REGION Network 24: Inicjacja parametrów nastwa zbirników z Modbus TCP
   RUNG wire#powerrail
      Move(in := "dbtags_Sterowanie"."Paramaetry _Zbiorniki".set_poziom_napełniania, out1 => "dbHold_RRG".set_poziom_napełniania)
      Move(in := "dbtags_Sterowanie"."Paramaetry _Zbiorniki".set_poziom_opróżniania, out1 => "dbHold_RRG".set_poziom_opróżniania)
      Move(in := "dbtags_Sterowanie"."Paramaetry _Zbiorniki".set_bity_sterowania_napęami_1, out1 => "dbHold_RRG".set_res_bity_sterowania_napęami_1)
      Move(in := "dbtags_Sterowanie"."Paramaetry _Zbiorniki".set_bity_sterowania_napęami_2, out1 => "dbHold_RRG".set_res_bity_sterowania_napęami_2)
      Move(in := "dbtags_Sterowanie"."Paramaetry _Zbiorniki".set_bity_tryb_napędów_1, out1 => "dbHold_RRG".set_res_bity_tryb_napędów_1)
      Move(in := "dbtags_Sterowanie"."Paramaetry _Zbiorniki".set_bity_tryb_napędów_2, out1 => "dbHold_RRG".set_res_bity_tryb_napędów_2)
   END_RUNG
   // the same network as SCL:
   "dbHold_RRG".set_poziom_napełniania := "dbtags_Sterowanie"."Paramaetry _Zbiorniki".set_poziom_napełniania;
   "dbHold_RRG".set_poziom_opróżniania := "dbtags_Sterowanie"."Paramaetry _Zbiorniki".set_poziom_opróżniania;
   "dbHold_RRG".set_res_bity_sterowania_napęami_1 := "dbtags_Sterowanie"."Paramaetry _Zbiorniki".set_bity_sterowania_napęami_1;
   "dbHold_RRG".set_res_bity_sterowania_napęami_2 := "dbtags_Sterowanie"."Paramaetry _Zbiorniki".set_bity_sterowania_napęami_2;
   "dbHold_RRG".set_res_bity_tryb_napędów_1 := "dbtags_Sterowanie"."Paramaetry _Zbiorniki".set_bity_tryb_napędów_1;
   "dbHold_RRG".set_res_bity_tryb_napędów_2 := "dbtags_Sterowanie"."Paramaetry _Zbiorniki".set_bity_tryb_napędów_2;
END_REGION

REGION Network 25
   RUNG wire#powerrail
      Move(in := "dbtags_Sterowanie"."Paramaetry _Zbiorniki".set_strategia_sterowania, out1 => "dbHold_RRG".set_strategia_sterowania)
      Move(in := "dbtags_Sterowanie"."Paramaetry _Zbiorniki".set_sterowanie_cyklem, out1 => "dbHold_RRG".set_sterowanie_cyklem)
      Move(in := "dbtags_Sterowanie"."Paramaetry _Zbiorniki".set_położenie_Z10, out1 => "dbHold_RRG".set_położenie_Z10)
   END_RUNG
   // the same network as SCL:
   "dbHold_RRG".set_strategia_sterowania := "dbtags_Sterowanie"."Paramaetry _Zbiorniki".set_strategia_sterowania;
   "dbHold_RRG".set_sterowanie_cyklem := "dbtags_Sterowanie"."Paramaetry _Zbiorniki".set_sterowanie_cyklem;
   "dbHold_RRG".set_położenie_Z10 := "dbtags_Sterowanie"."Paramaetry _Zbiorniki".set_położenie_Z10;
END_REGION

REGION Network 26: Napełnianie
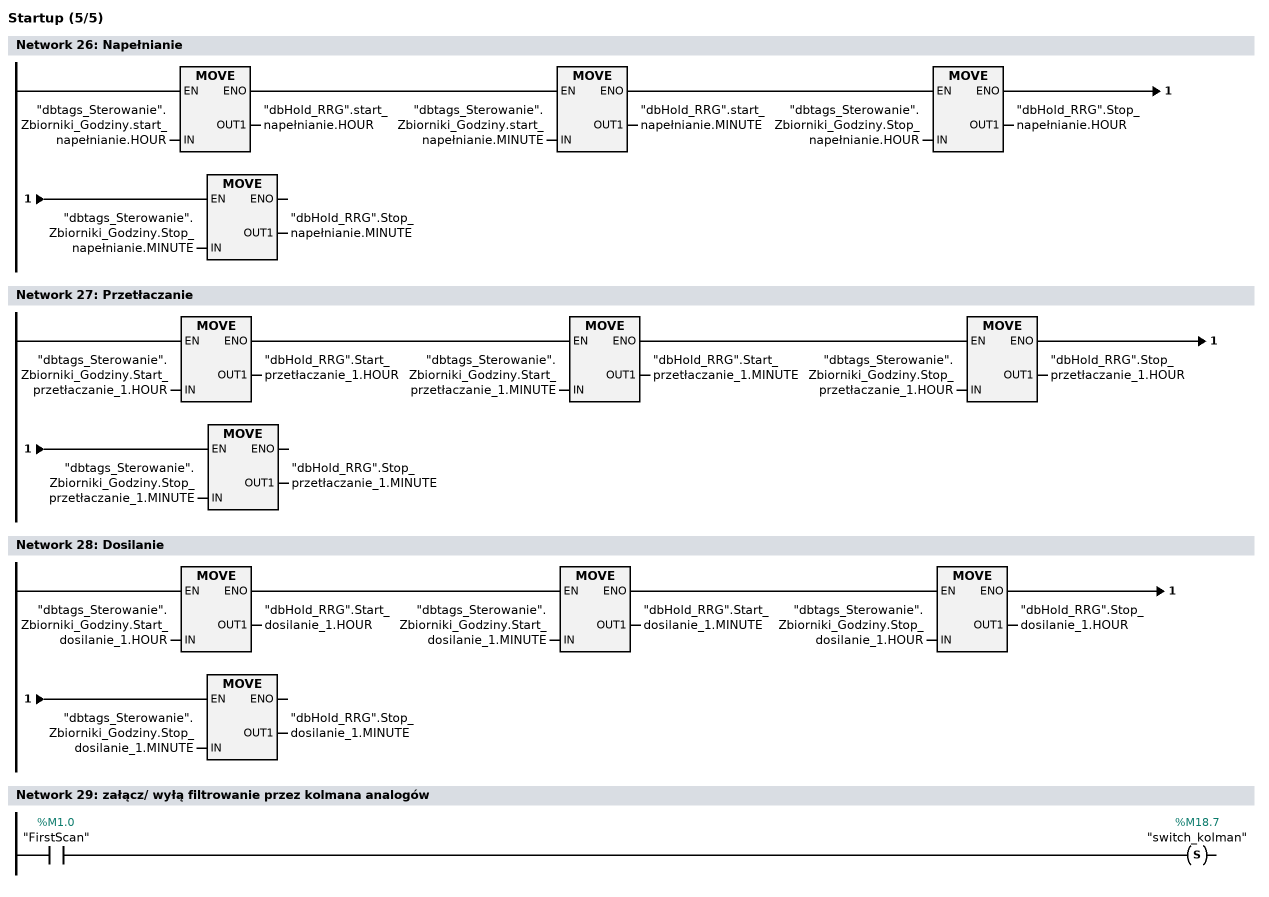
   RUNG wire#powerrail
      Move(in := "dbtags_Sterowanie".Zbiorniki_Godziny.start_napełnianie.HOUR, out1 => "dbHold_RRG".start_napełnianie.HOUR)
      Move(in := "dbtags_Sterowanie".Zbiorniki_Godziny.start_napełnianie.MINUTE, out1 => "dbHold_RRG".start_napełnianie.MINUTE)
      Move(in := "dbtags_Sterowanie".Zbiorniki_Godziny.Stop_napełnianie.HOUR, out1 => "dbHold_RRG".Stop_napełnianie.HOUR)
      Move(in := "dbtags_Sterowanie".Zbiorniki_Godziny.Stop_napełnianie.MINUTE, out1 => "dbHold_RRG".Stop_napełnianie.MINUTE)
   END_RUNG
   // the same network as SCL:
   "dbHold_RRG".start_napełnianie.HOUR := "dbtags_Sterowanie".Zbiorniki_Godziny.start_napełnianie.HOUR;
   "dbHold_RRG".start_napełnianie.MINUTE := "dbtags_Sterowanie".Zbiorniki_Godziny.start_napełnianie.MINUTE;
   "dbHold_RRG".Stop_napełnianie.HOUR := "dbtags_Sterowanie".Zbiorniki_Godziny.Stop_napełnianie.HOUR;
   "dbHold_RRG".Stop_napełnianie.MINUTE := "dbtags_Sterowanie".Zbiorniki_Godziny.Stop_napełnianie.MINUTE;
END_REGION

REGION Network 27: Przetłaczanie
   RUNG wire#powerrail
      Move(in := "dbtags_Sterowanie".Zbiorniki_Godziny.Start_przetłaczanie_1.HOUR, out1 => "dbHold_RRG".Start_przetłaczanie_1.HOUR)
      Move(in := "dbtags_Sterowanie".Zbiorniki_Godziny.Start_przetłaczanie_1.MINUTE, out1 => "dbHold_RRG".Start_przetłaczanie_1.MINUTE)
      Move(in := "dbtags_Sterowanie".Zbiorniki_Godziny.Stop_przetłaczanie_1.HOUR, out1 => "dbHold_RRG".Stop_przetłaczanie_1.HOUR)
      Move(in := "dbtags_Sterowanie".Zbiorniki_Godziny.Stop_przetłaczanie_1.MINUTE, out1 => "dbHold_RRG".Stop_przetłaczanie_1.MINUTE)
   END_RUNG
   // the same network as SCL:
   "dbHold_RRG".Start_przetłaczanie_1.HOUR := "dbtags_Sterowanie".Zbiorniki_Godziny.Start_przetłaczanie_1.HOUR;
   "dbHold_RRG".Start_przetłaczanie_1.MINUTE := "dbtags_Sterowanie".Zbiorniki_Godziny.Start_przetłaczanie_1.MINUTE;
   "dbHold_RRG".Stop_przetłaczanie_1.HOUR := "dbtags_Sterowanie".Zbiorniki_Godziny.Stop_przetłaczanie_1.HOUR;
   "dbHold_RRG".Stop_przetłaczanie_1.MINUTE := "dbtags_Sterowanie".Zbiorniki_Godziny.Stop_przetłaczanie_1.MINUTE;
END_REGION

REGION Network 28: Dosilanie
   RUNG wire#powerrail
      Move(in := "dbtags_Sterowanie".Zbiorniki_Godziny.Start_dosilanie_1.HOUR, out1 => "dbHold_RRG".Start_dosilanie_1.HOUR)
      Move(in := "dbtags_Sterowanie".Zbiorniki_Godziny.Start_dosilanie_1.MINUTE, out1 => "dbHold_RRG".Start_dosilanie_1.MINUTE)
      Move(in := "dbtags_Sterowanie".Zbiorniki_Godziny.Stop_dosilanie_1.HOUR, out1 => "dbHold_RRG".Stop_dosilanie_1.HOUR)
      Move(in := "dbtags_Sterowanie".Zbiorniki_Godziny.Stop_dosilanie_1.MINUTE, out1 => "dbHold_RRG".Stop_dosilanie_1.MINUTE)
   END_RUNG
   // the same network as SCL:
   "dbHold_RRG".Start_dosilanie_1.HOUR := "dbtags_Sterowanie".Zbiorniki_Godziny.Start_dosilanie_1.HOUR;
   "dbHold_RRG".Start_dosilanie_1.MINUTE := "dbtags_Sterowanie".Zbiorniki_Godziny.Start_dosilanie_1.MINUTE;
   "dbHold_RRG".Stop_dosilanie_1.HOUR := "dbtags_Sterowanie".Zbiorniki_Godziny.Stop_dosilanie_1.HOUR;
   "dbHold_RRG".Stop_dosilanie_1.MINUTE := "dbtags_Sterowanie".Zbiorniki_Godziny.Stop_dosilanie_1.MINUTE;
END_REGION

REGION Network 29: załącz/ wyłą filtrowanie przez kolmana analogów
   RUNG wire#powerrail
      Contact( "FirstScan" )
      S_Coil( "switch_kolman" )
   END_RUNG
   // the same network as SCL:
   IF "FirstScan" THEN "switch_kolman" := TRUE; END_IF;
END_REGION
END_ORGANIZATION_BLOCK

FUNCTION_BLOCK "Temp"   // FB22, LAD
{ S7_Optimized_Access := 'TRUE' }
VERSION : 0.1
// stored: AutoNumber true, IsIECCheckEnabled false, IsRetainMemResEnabled false, MemoryReserve 100, SetENOAutomatically false, UDAEnableTagReadback false
   VAR_INPUT
      Sub_PV_K1 : Real;   // Wspólczynnik pomniejszenia wyliczanego ciśnienia napotrzeby wyłączenia dodatowej pompy / Wspólczynnik pomniejszenia wyliczanego tlenu napotrzeby wyłączenia dodatowej dmuchawy
      InputWarning_H_PID { ExternalAccessible := 'False'; ExternalVisible := 'False'; ExternalWritable := 'False'} : Bool;   // Oszczerzenie górny limit
      InputWarning_L_PID { ExternalAccessible := 'False'; ExternalVisible := 'False'; ExternalWritable := 'False'} : Bool;   // Oczszczerzenie dolny limit
   END_VAR
   VAR_IN_OUT
      Set_K1 { ExternalWritable := 'False'} : Bool;   // Dostaw 1 dodatkową / Dostaw 1 dmuchawę dodatkową
   END_VAR
   VAR_TEMP
      Temp_SV_Int : Int;
   END_VAR
   VAR_TEMP   // added for the SCL form of the ladder/FBD networks
      _w1 : Bool;
      _w2 : Bool;
   END_VAR
BEGIN

REGION Network 1
   // OB 30 Network 14
END_REGION

REGION Network 2: Przekazanie wartości na wyjście analogowe "Out_Hz" -
   // Jeśli znacznik TmP_Set_SV (tymczasowe ustawienie Hz) wyłączony to na wyjście QW90 przekazywana jest wartość wyliczona z PID
   // Jeśli znacznik Tmp_Set_SV jest True to na wyjście przekazywana jest wartość tymczasowa 30Hz
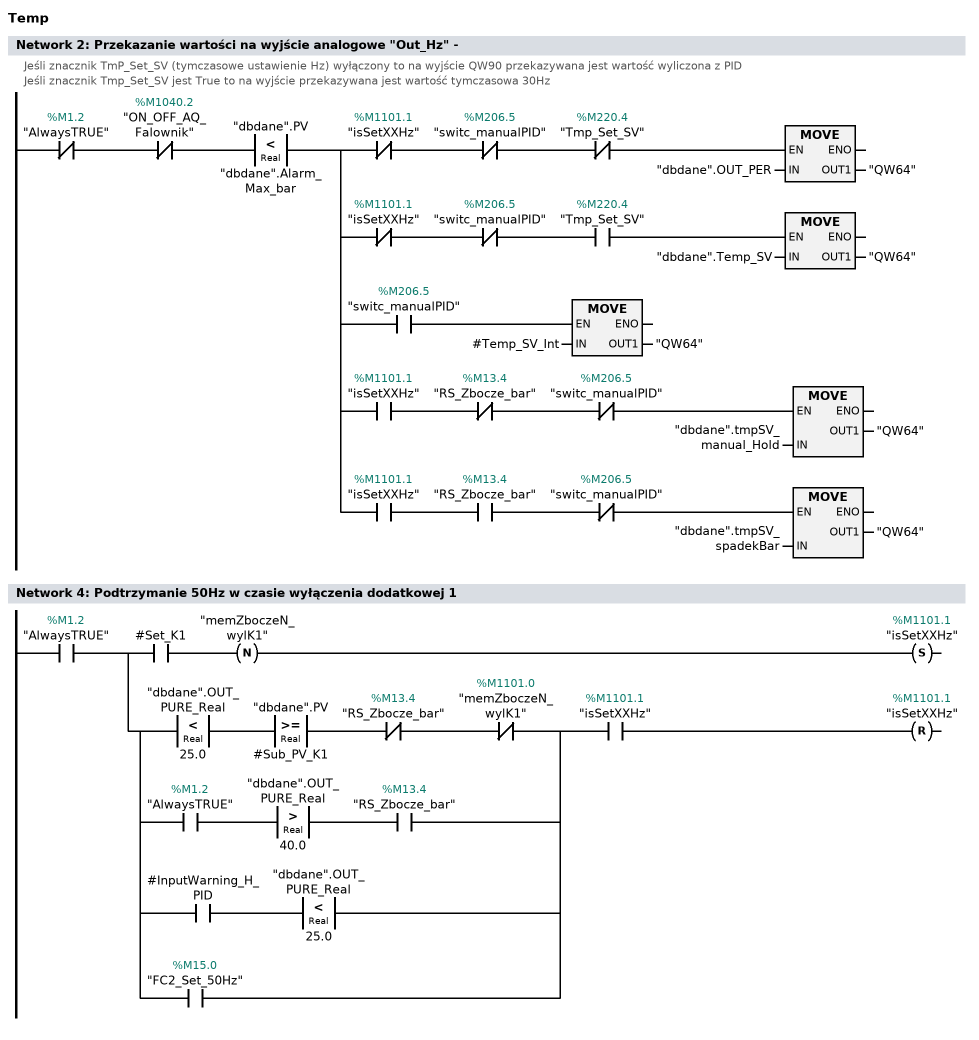
   RUNG wire#powerrail
      I_Contact( "AlwaysTRUE" )
      I_Contact( "ON_OFF_AQ_Falownik" )
      { S7_Templates := "SrcType := Real" } LT_Contact(in1 := "dbdane".PV, in2 := "dbdane".Alarm_Max_bar)
      wire#w1
      I_Contact( "isSetXXHz" )
      I_Contact( "switc_manualPID" )
      I_Contact( "Tmp_Set_SV" )
      { S7_GenerateENO := "TRUE" } Move(in := "dbdane".OUT_PER, out1 => "QW64")
   END_RUNG
   RUNG wire#w1
      I_Contact( "isSetXXHz" )
      I_Contact( "switc_manualPID" )
      Contact( "Tmp_Set_SV" )
      { S7_GenerateENO := "TRUE" } Move(in := "dbdane".Temp_SV, out1 => "QW64")
   END_RUNG
   RUNG wire#w1
      Contact( "switc_manualPID" )
      { S7_GenerateENO := "TRUE" } Move(in := #Temp_SV_Int, out1 => "QW64")
   END_RUNG
   RUNG wire#w1
      Contact( "isSetXXHz" )
      I_Contact( "RS_Zbocze_bar" )
      I_Contact( "switc_manualPID" )
      { S7_GenerateENO := "TRUE" } Move(in := "dbdane".tmpSV_manual_Hold, out1 => "QW64")
   END_RUNG
   RUNG wire#w1
      Contact( "isSetXXHz" )
      Contact( "RS_Zbocze_bar" )
      I_Contact( "switc_manualPID" )
      { S7_GenerateENO := "TRUE" } Move(in := "dbdane".tmpSV_spadekBar, out1 => "QW64")
   END_RUNG
   // the same network as SCL:
   #_w1 := NOT "AlwaysTRUE" AND NOT "ON_OFF_AQ_Falownik" AND ("dbdane".PV < "dbdane".Alarm_Max_bar);
   IF #_w1 AND NOT "isSetXXHz" AND NOT "switc_manualPID" AND NOT "Tmp_Set_SV" THEN
       "QW64" := "dbdane".OUT_PER;
   END_IF;
   IF #_w1 AND NOT "isSetXXHz" AND NOT "switc_manualPID" AND "Tmp_Set_SV" THEN
       "QW64" := "dbdane".Temp_SV;
   END_IF;
   IF #_w1 AND "switc_manualPID" THEN "QW64" := #Temp_SV_Int; END_IF;
   IF #_w1 AND "isSetXXHz" AND NOT "RS_Zbocze_bar" AND NOT "switc_manualPID" THEN
       "QW64" := "dbdane".tmpSV_manual_Hold;
   END_IF;
   IF #_w1 AND "isSetXXHz" AND "RS_Zbocze_bar" AND NOT "switc_manualPID" THEN
       "QW64" := "dbdane".tmpSV_spadekBar;
   END_IF;
END_REGION

REGION Network 3: FB1 Network 22
END_REGION

REGION Network 4: Podtrzymanie 50Hz w czasie wyłączenia dodatkowej 1
   RUNG wire#powerrail
      Contact( "AlwaysTRUE" )
      wire#w1
      Contact( #Set_K1 )
      N_Trig( "memZboczeN_wylK1" )
      S_Coil( "isSetXXHz" )
   END_RUNG
   RUNG wire#w1
      { S7_Templates := "SrcType := Real" } LT_Contact(in1 := "dbdane".OUT_PURE_Real, in2 := 25.0)
      { S7_Templates := "SrcType := Real" } GE_Contact(in1 := "dbdane".PV, in2 := #Sub_PV_K1)
      I_Contact( "RS_Zbocze_bar" )
      I_Contact( "memZboczeN_wylK1" )
      wire#w2
      Contact( "isSetXXHz" )
      R_Coil( "isSetXXHz" )
   END_RUNG
   RUNG wire#w1
      Contact( "AlwaysTRUE" )
      { S7_Templates := "SrcType := Real" } GT_Contact(in1 := "dbdane".OUT_PURE_Real, in2 := 40.0)
      Contact( "RS_Zbocze_bar" )
   END_RUNG wire#w2
   RUNG wire#w1
      Contact( #InputWarning_H_PID )
      { S7_Templates := "SrcType := Real" } LT_Contact(in1 := "dbdane".OUT_PURE_Real, in2 := 25.0)
   END_RUNG wire#w2
   RUNG wire#w1
      Contact( "FC2_Set_50Hz" )
   END_RUNG wire#w2
   // the same network as SCL:
   #_w1 := "AlwaysTRUE" AND #Set_K1;
   #_w2 := NOT #_w1 AND "memZboczeN_wylK1";   // falling edge
   "memZboczeN_wylK1" := #_w1;
   IF #_w2 THEN "isSetXXHz" := TRUE; END_IF;
   IF "AlwaysTRUE" AND ((("dbdane".OUT_PURE_Real < 25.0) AND ("dbdane".PV >= #Sub_PV_K1) AND NOT "RS_Zbocze_bar" AND NOT "memZboczeN_wylK1") OR ("AlwaysTRUE" AND ("dbdane".OUT_PURE_Real > 40.0) AND "RS_Zbocze_bar") OR (#InputWarning_H_PID AND ("dbdane".OUT_PURE_Real < 25.0)) OR "FC2_Set_50Hz") AND "isSetXXHz" THEN
       "isSetXXHz" := FALSE;
   END_IF;
END_REGION
END_FUNCTION_BLOCK

FUNCTION_BLOCK "WatchDog PLC - WinCC"   // FB13, LAD
TITLE = WatchDog PLC - WinCC
{ S7_Optimized_Access := 'TRUE' }
AUTHOR : rtecmer
VERSION : 0.1
// Kontrola komunikacji PLC z WinCC SCADA . Zerwanie komunikacji przekazywane do WinCC SCADA i PLC Master S7-300 (RS3)
// stored: AutoNumber true, IsIECCheckEnabled false, IsRetainMemResEnabled false, MemoryReserve 500, SetENOAutomatically false, UDAEnableTagReadback false
   VAR_TEMP   // added for the SCL form of the ladder/FBD networks
      _w1 : Bool;
      _w2 : Bool;
   END_VAR
BEGIN

REGION Network 1: WatchDog WinCC - PLC
   // Konfiguracja WinCC Flexible - ustawiony Area Point (Coordination) na DB29 DBW12
   // WinCC wpisuje z częstotliwością 0,9s na zmianę wartości 1 i 5.
   // PLC  kontroluje tę zmianę poprzez Timer TON z histerezą 10s. Jeśli nastąpi przerwanie komunikacji
   // zasygnalizuje to jeden z dwóch TON ustawiając możliwość inkrementacji zmiennej pomocniczej w instancji "Dane_ComunicationControlHMI".tempWatchDog_WinCC i ustawi bitu alarmu braku komunikacji z WinCC  
   // Po powrocie komunikacji zmienna "Dane_ComunicationControlHMI".tempWatchDog_WinCC jest zerowana.
   // Wartośc zmiennej  "Dane_ComunicationControlHMI".tempWatchDog_WinCC jest pobierana przez scipt VB WinCC jeśli jest 0 to comunikacja OK jeśli natomiast  > 0 to script VB inkrementuje wewnętrzną zmienną i ustawia alarm w WinCC.
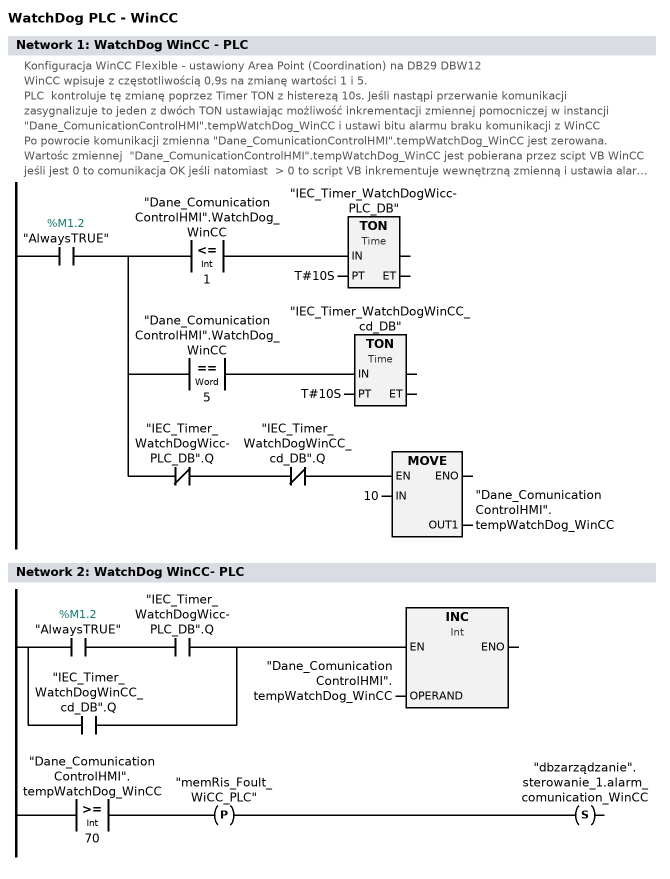
   RUNG wire#powerrail
      Contact( "AlwaysTRUE" )
      wire#w1
      { S7_Templates := "SrcType := Int" } LE_Contact(in1 := "Dane_ComunicationControlHMI".WatchDog_WinCC, in2 := 1)
      { S7_Templates := "time_type := Time" } "IEC_Timer_WatchDogWicc-PLC_DB".TON(pt := T#10S, et =>)
   END_RUNG
   RUNG wire#w1
      { S7_Templates := "SrcType := Word" } EQ_Contact(in1 := "Dane_ComunicationControlHMI".WatchDog_WinCC, in2 := 5)
      { S7_Templates := "time_type := Time" } "IEC_Timer_WatchDogWinCC_cd_DB".TON(pt := T#10S, et =>)
   END_RUNG
   RUNG wire#w1
      I_Contact( "IEC_Timer_WatchDogWicc-PLC_DB".Q )
      I_Contact( "IEC_Timer_WatchDogWinCC_cd_DB".Q )
      Move(in := 10, out1 => "Dane_ComunicationControlHMI".tempWatchDog_WinCC)
   END_RUNG
   // the same network as SCL:
   "IEC_Timer_WatchDogWicc-PLC_DB".TON(IN := "AlwaysTRUE" AND ("Dane_ComunicationControlHMI".WatchDog_WinCC <= 1),
                           PT := T#10S);
   "IEC_Timer_WatchDogWinCC_cd_DB".TON(IN := "AlwaysTRUE" AND ("Dane_ComunicationControlHMI".WatchDog_WinCC = 5),
                           PT := T#10S);
   IF "AlwaysTRUE" AND NOT "IEC_Timer_WatchDogWicc-PLC_DB".Q AND NOT "IEC_Timer_WatchDogWinCC_cd_DB".Q THEN
       "Dane_ComunicationControlHMI".tempWatchDog_WinCC := 10;
   END_IF;
END_REGION

REGION Network 2: WatchDog WinCC- PLC
   RUNG wire#powerrail
      Contact( "AlwaysTRUE" )
      Contact( "IEC_Timer_WatchDogWicc-PLC_DB".Q )
      wire#w1
      { S7_Templates := "DestType := Int" } Inc( "Dane_ComunicationControlHMI".tempWatchDog_WinCC )
   END_RUNG
   RUNG wire#powerrail
      Contact( "IEC_Timer_WatchDogWinCC_cd_DB".Q )
   END_RUNG wire#w1
   RUNG wire#powerrail
      { S7_Templates := "SrcType := Int" } GE_Contact(in1 := "Dane_ComunicationControlHMI".tempWatchDog_WinCC, in2 := 70)
      P_Trig( "memRis_Foult_WiCC_PLC" )
      S_Coil( "dbzarządzanie".sterowanie_1.alarm_comunication_WinCC )
   END_RUNG
   // the same network as SCL:
   IF ("AlwaysTRUE" AND "IEC_Timer_WatchDogWicc-PLC_DB".Q) OR "IEC_Timer_WatchDogWinCC_cd_DB".Q THEN
       "Dane_ComunicationControlHMI".tempWatchDog_WinCC := "Dane_ComunicationControlHMI".tempWatchDog_WinCC + 1;
   END_IF;
   #_w1 := "Dane_ComunicationControlHMI".tempWatchDog_WinCC >= 70;
   #_w2 := #_w1 AND NOT "memRis_Foult_WiCC_PLC";   // rising edge
   "memRis_Foult_WiCC_PLC" := #_w1;
   IF #_w2 THEN "dbzarządzanie".sterowanie_1.alarm_comunication_WinCC := TRUE; END_IF;
END_REGION
END_FUNCTION_BLOCK

FUNCTION "MPP04_2_rez" : Void   // FC24, LAD
TITLE = Read data from SC100
{ S7_Optimized_Access := 'TRUE' }
AUTHOR : rtecmer
VERSION : 0.1
// Czytanie z SC1000 
// Obsługa protokołu Master Modbus RTU.  Odczyt pomiarów  i status czujnika SC1000
// stored: AutoNumber false, IsIECCheckEnabled false, SetENOAutomatically false, UDAEnableTagReadback false
   VAR_TEMP
      Wielkość_przeływu_Adres0_0 : DWord;
      Wielkość_przeływu_Adres0_1 : DWord;
      Wielkość_przeływu_Adres2_0 : DWord;
      Wielkość_przeływu_Adres2_2 : DWord;
   END_VAR
   VAR_TEMP   // added for the SCL form of the ladder/FBD networks
      _w1 : Bool;
      _w2 : Bool;
   END_VAR
BEGIN

REGION Network 1
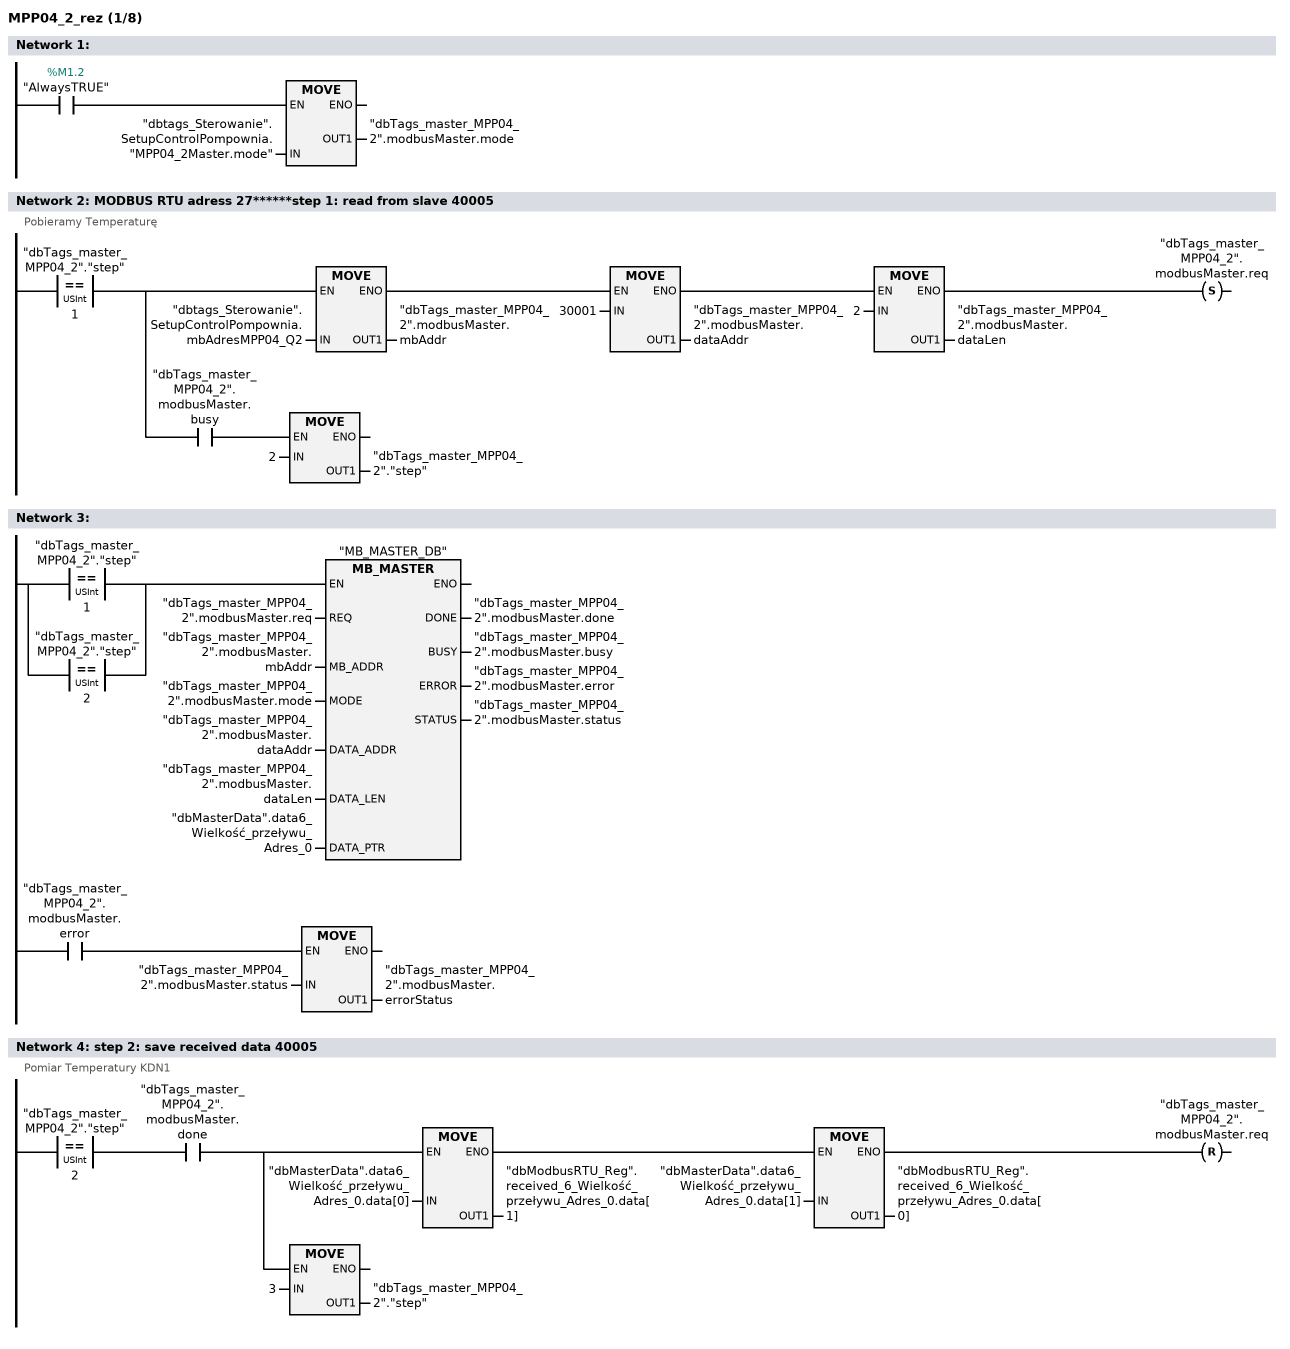
   RUNG wire#powerrail
      Contact( "AlwaysTRUE" )
      { S7_GenerateENO := "TRUE" } Move(in := "dbtags_Sterowanie".SetupControlPompownia."MPP04_2Master.mode", out1 => "dbTags_master_MPP04_2".modbusMaster.mode)
   END_RUNG
   // the same network as SCL:
   IF "AlwaysTRUE" THEN
       "dbTags_master_MPP04_2".modbusMaster.mode := "dbtags_Sterowanie".SetupControlPompownia."MPP04_2Master.mode";
   END_IF;
END_REGION

REGION Network 2: MODBUS RTU adress 27******step 1: read from slave 40005
   // Pobieramy Temperaturę
   RUNG wire#powerrail
      { S7_Templates := "SrcType := USInt" } EQ_Contact(in1 := "dbTags_master_MPP04_2"."step", in2 := 1)
      wire#w1
      Move(in := "dbtags_Sterowanie".SetupControlPompownia.mbAdresMPP04_Q2, out1 => "dbTags_master_MPP04_2".modbusMaster.mbAddr)
      { S7_GenerateENO := "TRUE" } Move(in := 30001, out1 => "dbTags_master_MPP04_2".modbusMaster.dataAddr)
      Move(in := 2, out1 => "dbTags_master_MPP04_2".modbusMaster.dataLen)
      S_Coil( "dbTags_master_MPP04_2".modbusMaster.req )
   END_RUNG
   RUNG wire#w1
      Contact( "dbTags_master_MPP04_2".modbusMaster.busy )
      { S7_GenerateENO := "TRUE" } Move(in := 2, out1 => "dbTags_master_MPP04_2"."step")
   END_RUNG
   // the same network as SCL:
   // ENO of a box is taken as its EN; it also drops when the box reports an error
   #_w1 := "dbTags_master_MPP04_2"."step" = 1;
   IF #_w1 THEN
       "dbTags_master_MPP04_2".modbusMaster.mbAddr := "dbtags_Sterowanie".SetupControlPompownia.mbAdresMPP04_Q2;
       "dbTags_master_MPP04_2".modbusMaster.dataAddr := 30001;
       "dbTags_master_MPP04_2".modbusMaster.dataLen := 2;
       "dbTags_master_MPP04_2".modbusMaster.req := TRUE;
   END_IF;
   IF #_w1 AND "dbTags_master_MPP04_2".modbusMaster.busy THEN "dbTags_master_MPP04_2"."step" := 2; END_IF;
END_REGION

REGION Network 3
   RUNG wire#powerrail
      { S7_Templates := "SrcType := USInt" } EQ_Contact(in1 := "dbTags_master_MPP04_2"."step", in2 := 1)
      wire#w1
      "MB_MASTER_DB".MB_MASTER(REQ := "dbTags_master_MPP04_2".modbusMaster.req, MB_ADDR := "dbTags_master_MPP04_2".modbusMaster.mbAddr, MODE := "dbTags_master_MPP04_2".modbusMaster.mode, DATA_ADDR := "dbTags_master_MPP04_2".modbusMaster.dataAddr, DATA_LEN := "dbTags_master_MPP04_2".modbusMaster.dataLen, DATA_PTR := "dbMasterData".data6_Wielkość_przeływu_Adres_0, DONE => "dbTags_master_MPP04_2".modbusMaster.done, BUSY => "dbTags_master_MPP04_2".modbusMaster.busy, ERROR => "dbTags_master_MPP04_2".modbusMaster.error, STATUS => "dbTags_master_MPP04_2".modbusMaster.status)
   END_RUNG
   RUNG wire#powerrail
      { S7_Templates := "SrcType := USInt" } EQ_Contact(in1 := "dbTags_master_MPP04_2"."step", in2 := 2)
   END_RUNG wire#w1
   RUNG wire#powerrail
      Contact( "dbTags_master_MPP04_2".modbusMaster.error )
      { S7_GenerateENO := "TRUE" } Move(in := "dbTags_master_MPP04_2".modbusMaster.status, out1 => "dbTags_master_MPP04_2".modbusMaster.errorStatus)
   END_RUNG
   // the same network as SCL:
   IF ("dbTags_master_MPP04_2"."step" = 1) OR ("dbTags_master_MPP04_2"."step" = 2) THEN
       "MB_MASTER_DB"(REQ := "dbTags_master_MPP04_2".modbusMaster.req,   // MB_MASTER
                      MB_ADDR := "dbTags_master_MPP04_2".modbusMaster.mbAddr,
                      MODE := "dbTags_master_MPP04_2".modbusMaster.mode,
                      DATA_ADDR := "dbTags_master_MPP04_2".modbusMaster.dataAddr,
                      DATA_LEN := "dbTags_master_MPP04_2".modbusMaster.dataLen,
                      DATA_PTR := "dbMasterData".data6_Wielkość_przeływu_Adres_0,
                      DONE => "dbTags_master_MPP04_2".modbusMaster.done,
                      BUSY => "dbTags_master_MPP04_2".modbusMaster.busy,
                      ERROR => "dbTags_master_MPP04_2".modbusMaster.error,
                      STATUS => "dbTags_master_MPP04_2".modbusMaster.status);
   END_IF;
   IF "dbTags_master_MPP04_2".modbusMaster.error THEN
       "dbTags_master_MPP04_2".modbusMaster.errorStatus := "dbTags_master_MPP04_2".modbusMaster.status;
   END_IF;
END_REGION

REGION Network 4: step 2: save received data 40005
   // Pomiar Temperatury KDN1
   RUNG wire#powerrail
      { S7_Templates := "SrcType := USInt" } EQ_Contact(in1 := "dbTags_master_MPP04_2"."step", in2 := 2)
      Contact( "dbTags_master_MPP04_2".modbusMaster.done )
      wire#w1
      { S7_GenerateENO := "TRUE" } Move(in := "dbMasterData".data6_Wielkość_przeływu_Adres_0.data[0], out1 => "dbModbusRTU_Reg".received_6_Wielkość_przeływu_Adres_0.data[1])
      { S7_GenerateENO := "TRUE" } Move(in := "dbMasterData".data6_Wielkość_przeływu_Adres_0.data[1], out1 => "dbModbusRTU_Reg".received_6_Wielkość_przeływu_Adres_0.data[0])
      R_Coil( "dbTags_master_MPP04_2".modbusMaster.req )
   END_RUNG
   RUNG wire#w1
      { S7_GenerateENO := "TRUE" } Move(in := 3, out1 => "dbTags_master_MPP04_2"."step")
   END_RUNG
   // the same network as SCL:
   // ENO of a box is taken as its EN; it also drops when the box reports an error
   IF ("dbTags_master_MPP04_2"."step" = 2) AND "dbTags_master_MPP04_2".modbusMaster.done THEN
       "dbModbusRTU_Reg".received_6_Wielkość_przeływu_Adres_0.data[1] := "dbMasterData".data6_Wielkość_przeływu_Adres_0.data[0];
       "dbModbusRTU_Reg".received_6_Wielkość_przeływu_Adres_0.data[0] := "dbMasterData".data6_Wielkość_przeływu_Adres_0.data[1];
       "dbTags_master_MPP04_2".modbusMaster.req := FALSE;
       "dbTags_master_MPP04_2"."step" := 3;
   END_IF;
END_REGION

REGION Network 5: MODBUS RTU adress 27******step 3: read from slave 40001
   // Bytes Error
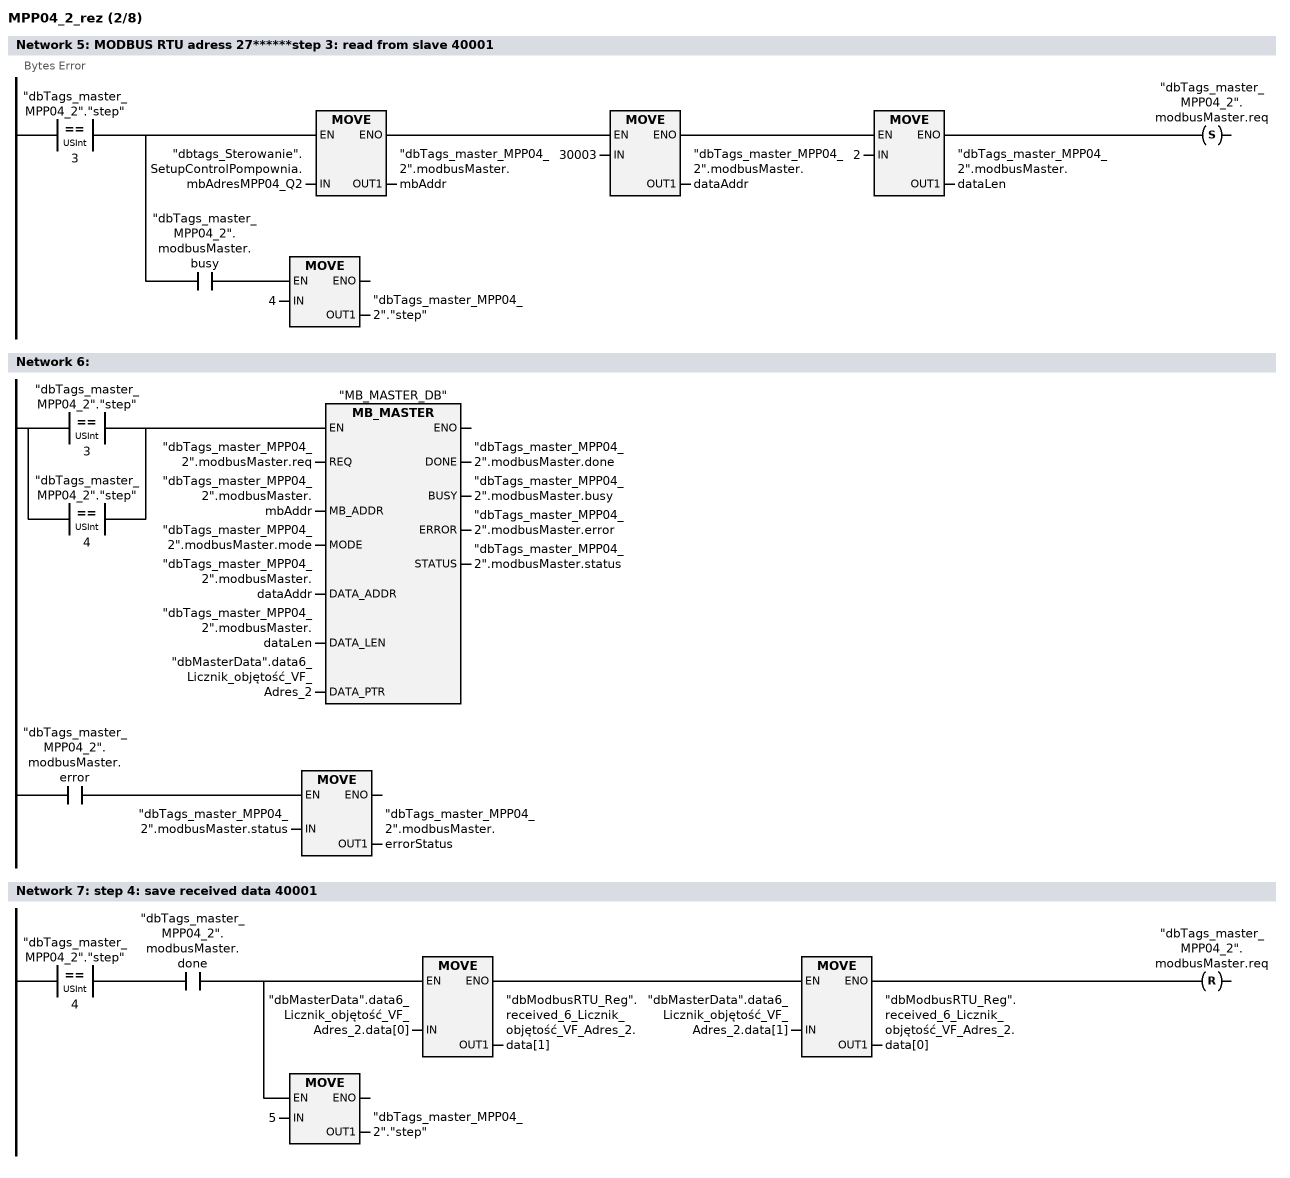
   RUNG wire#powerrail
      { S7_Templates := "SrcType := USInt" } EQ_Contact(in1 := "dbTags_master_MPP04_2"."step", in2 := 3)
      wire#w1
      Move(in := "dbtags_Sterowanie".SetupControlPompownia.mbAdresMPP04_Q2, out1 => "dbTags_master_MPP04_2".modbusMaster.mbAddr)
      { S7_GenerateENO := "TRUE" } Move(in := 30003, out1 => "dbTags_master_MPP04_2".modbusMaster.dataAddr)
      Move(in := 2, out1 => "dbTags_master_MPP04_2".modbusMaster.dataLen)
      S_Coil( "dbTags_master_MPP04_2".modbusMaster.req )
   END_RUNG
   RUNG wire#w1
      Contact( "dbTags_master_MPP04_2".modbusMaster.busy )
      { S7_GenerateENO := "TRUE" } Move(in := 4, out1 => "dbTags_master_MPP04_2"."step")
   END_RUNG
   // the same network as SCL:
   // ENO of a box is taken as its EN; it also drops when the box reports an error
   #_w1 := "dbTags_master_MPP04_2"."step" = 3;
   IF #_w1 THEN
       "dbTags_master_MPP04_2".modbusMaster.mbAddr := "dbtags_Sterowanie".SetupControlPompownia.mbAdresMPP04_Q2;
       "dbTags_master_MPP04_2".modbusMaster.dataAddr := 30003;
       "dbTags_master_MPP04_2".modbusMaster.dataLen := 2;
       "dbTags_master_MPP04_2".modbusMaster.req := TRUE;
   END_IF;
   IF #_w1 AND "dbTags_master_MPP04_2".modbusMaster.busy THEN "dbTags_master_MPP04_2"."step" := 4; END_IF;
END_REGION

REGION Network 6
   RUNG wire#powerrail
      { S7_Templates := "SrcType := USInt" } EQ_Contact(in1 := "dbTags_master_MPP04_2"."step", in2 := 3)
      wire#w1
      "MB_MASTER_DB".MB_MASTER(REQ := "dbTags_master_MPP04_2".modbusMaster.req, MB_ADDR := "dbTags_master_MPP04_2".modbusMaster.mbAddr, MODE := "dbTags_master_MPP04_2".modbusMaster.mode, DATA_ADDR := "dbTags_master_MPP04_2".modbusMaster.dataAddr, DATA_LEN := "dbTags_master_MPP04_2".modbusMaster.dataLen, DATA_PTR := "dbMasterData".data6_Licznik_objętość_VF_Adres_2, DONE => "dbTags_master_MPP04_2".modbusMaster.done, BUSY => "dbTags_master_MPP04_2".modbusMaster.busy, ERROR => "dbTags_master_MPP04_2".modbusMaster.error, STATUS => "dbTags_master_MPP04_2".modbusMaster.status)
   END_RUNG
   RUNG wire#powerrail
      { S7_Templates := "SrcType := USInt" } EQ_Contact(in1 := "dbTags_master_MPP04_2"."step", in2 := 4)
   END_RUNG wire#w1
   RUNG wire#powerrail
      Contact( "dbTags_master_MPP04_2".modbusMaster.error )
      { S7_GenerateENO := "TRUE" } Move(in := "dbTags_master_MPP04_2".modbusMaster.status, out1 => "dbTags_master_MPP04_2".modbusMaster.errorStatus)
   END_RUNG
   // the same network as SCL:
   IF ("dbTags_master_MPP04_2"."step" = 3) OR ("dbTags_master_MPP04_2"."step" = 4) THEN
       "MB_MASTER_DB"(REQ := "dbTags_master_MPP04_2".modbusMaster.req,   // MB_MASTER
                      MB_ADDR := "dbTags_master_MPP04_2".modbusMaster.mbAddr,
                      MODE := "dbTags_master_MPP04_2".modbusMaster.mode,
                      DATA_ADDR := "dbTags_master_MPP04_2".modbusMaster.dataAddr,
                      DATA_LEN := "dbTags_master_MPP04_2".modbusMaster.dataLen,
                      DATA_PTR := "dbMasterData".data6_Licznik_objętość_VF_Adres_2,
                      DONE => "dbTags_master_MPP04_2".modbusMaster.done,
                      BUSY => "dbTags_master_MPP04_2".modbusMaster.busy,
                      ERROR => "dbTags_master_MPP04_2".modbusMaster.error,
                      STATUS => "dbTags_master_MPP04_2".modbusMaster.status);
   END_IF;
   IF "dbTags_master_MPP04_2".modbusMaster.error THEN
       "dbTags_master_MPP04_2".modbusMaster.errorStatus := "dbTags_master_MPP04_2".modbusMaster.status;
   END_IF;
END_REGION

REGION Network 7: step 4: save received data 40001
   RUNG wire#powerrail
      { S7_Templates := "SrcType := USInt" } EQ_Contact(in1 := "dbTags_master_MPP04_2"."step", in2 := 4)
      Contact( "dbTags_master_MPP04_2".modbusMaster.done )
      wire#w1
      { S7_GenerateENO := "TRUE" } Move(in := "dbMasterData".data6_Licznik_objętość_VF_Adres_2.data[0], out1 => "dbModbusRTU_Reg".received_6_Licznik_objętość_VF_Adres_2.data[1])
      { S7_GenerateENO := "TRUE" } Move(in := "dbMasterData".data6_Licznik_objętość_VF_Adres_2.data[1], out1 => "dbModbusRTU_Reg".received_6_Licznik_objętość_VF_Adres_2.data[0])
      R_Coil( "dbTags_master_MPP04_2".modbusMaster.req )
   END_RUNG
   RUNG wire#w1
      { S7_GenerateENO := "TRUE" } Move(in := 5, out1 => "dbTags_master_MPP04_2"."step")
   END_RUNG
   // the same network as SCL:
   // ENO of a box is taken as its EN; it also drops when the box reports an error
   IF ("dbTags_master_MPP04_2"."step" = 4) AND "dbTags_master_MPP04_2".modbusMaster.done THEN
       "dbModbusRTU_Reg".received_6_Licznik_objętość_VF_Adres_2.data[1] := "dbMasterData".data6_Licznik_objętość_VF_Adres_2.data[0];
       "dbModbusRTU_Reg".received_6_Licznik_objętość_VF_Adres_2.data[0] := "dbMasterData".data6_Licznik_objętość_VF_Adres_2.data[1];
       "dbTags_master_MPP04_2".modbusMaster.req := FALSE;
       "dbTags_master_MPP04_2"."step" := 5;
   END_IF;
END_REGION

REGION Network 8: MODBUS RTU adress 27******step 5: read from slave 40002
   // Pobieramy status sondy
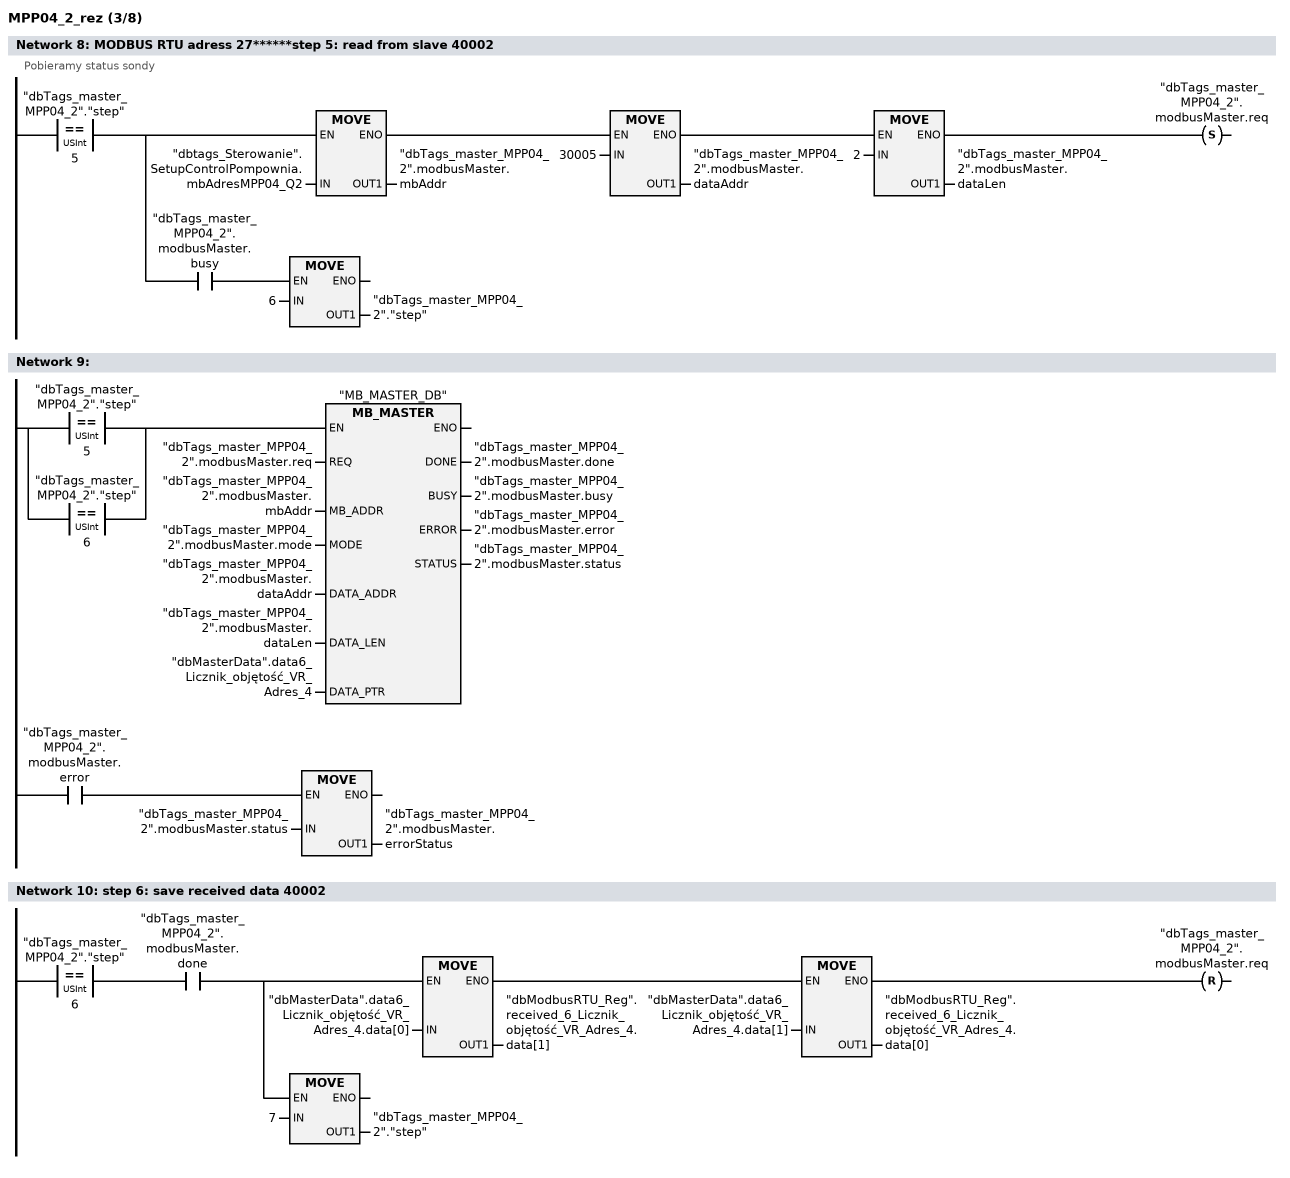
   RUNG wire#powerrail
      { S7_Templates := "SrcType := USInt" } EQ_Contact(in1 := "dbTags_master_MPP04_2"."step", in2 := 5)
      wire#w1
      Move(in := "dbtags_Sterowanie".SetupControlPompownia.mbAdresMPP04_Q2, out1 => "dbTags_master_MPP04_2".modbusMaster.mbAddr)
      { S7_GenerateENO := "TRUE" } Move(in := 30005, out1 => "dbTags_master_MPP04_2".modbusMaster.dataAddr)
      Move(in := 2, out1 => "dbTags_master_MPP04_2".modbusMaster.dataLen)
      S_Coil( "dbTags_master_MPP04_2".modbusMaster.req )
   END_RUNG
   RUNG wire#w1
      Contact( "dbTags_master_MPP04_2".modbusMaster.busy )
      { S7_GenerateENO := "TRUE" } Move(in := 6, out1 => "dbTags_master_MPP04_2"."step")
   END_RUNG
   // the same network as SCL:
   // ENO of a box is taken as its EN; it also drops when the box reports an error
   #_w1 := "dbTags_master_MPP04_2"."step" = 5;
   IF #_w1 THEN
       "dbTags_master_MPP04_2".modbusMaster.mbAddr := "dbtags_Sterowanie".SetupControlPompownia.mbAdresMPP04_Q2;
       "dbTags_master_MPP04_2".modbusMaster.dataAddr := 30005;
       "dbTags_master_MPP04_2".modbusMaster.dataLen := 2;
       "dbTags_master_MPP04_2".modbusMaster.req := TRUE;
   END_IF;
   IF #_w1 AND "dbTags_master_MPP04_2".modbusMaster.busy THEN "dbTags_master_MPP04_2"."step" := 6; END_IF;
END_REGION

REGION Network 9
   RUNG wire#powerrail
      { S7_Templates := "SrcType := USInt" } EQ_Contact(in1 := "dbTags_master_MPP04_2"."step", in2 := 5)
      wire#w1
      "MB_MASTER_DB".MB_MASTER(REQ := "dbTags_master_MPP04_2".modbusMaster.req, MB_ADDR := "dbTags_master_MPP04_2".modbusMaster.mbAddr, MODE := "dbTags_master_MPP04_2".modbusMaster.mode, DATA_ADDR := "dbTags_master_MPP04_2".modbusMaster.dataAddr, DATA_LEN := "dbTags_master_MPP04_2".modbusMaster.dataLen, DATA_PTR := "dbMasterData".data6_Licznik_objętość_VR_Adres_4, DONE => "dbTags_master_MPP04_2".modbusMaster.done, BUSY => "dbTags_master_MPP04_2".modbusMaster.busy, ERROR => "dbTags_master_MPP04_2".modbusMaster.error, STATUS => "dbTags_master_MPP04_2".modbusMaster.status)
   END_RUNG
   RUNG wire#powerrail
      { S7_Templates := "SrcType := USInt" } EQ_Contact(in1 := "dbTags_master_MPP04_2"."step", in2 := 6)
   END_RUNG wire#w1
   RUNG wire#powerrail
      Contact( "dbTags_master_MPP04_2".modbusMaster.error )
      { S7_GenerateENO := "TRUE" } Move(in := "dbTags_master_MPP04_2".modbusMaster.status, out1 => "dbTags_master_MPP04_2".modbusMaster.errorStatus)
   END_RUNG
   // the same network as SCL:
   IF ("dbTags_master_MPP04_2"."step" = 5) OR ("dbTags_master_MPP04_2"."step" = 6) THEN
       "MB_MASTER_DB"(REQ := "dbTags_master_MPP04_2".modbusMaster.req,   // MB_MASTER
                      MB_ADDR := "dbTags_master_MPP04_2".modbusMaster.mbAddr,
                      MODE := "dbTags_master_MPP04_2".modbusMaster.mode,
                      DATA_ADDR := "dbTags_master_MPP04_2".modbusMaster.dataAddr,
                      DATA_LEN := "dbTags_master_MPP04_2".modbusMaster.dataLen,
                      DATA_PTR := "dbMasterData".data6_Licznik_objętość_VR_Adres_4,
                      DONE => "dbTags_master_MPP04_2".modbusMaster.done,
                      BUSY => "dbTags_master_MPP04_2".modbusMaster.busy,
                      ERROR => "dbTags_master_MPP04_2".modbusMaster.error,
                      STATUS => "dbTags_master_MPP04_2".modbusMaster.status);
   END_IF;
   IF "dbTags_master_MPP04_2".modbusMaster.error THEN
       "dbTags_master_MPP04_2".modbusMaster.errorStatus := "dbTags_master_MPP04_2".modbusMaster.status;
   END_IF;
END_REGION

REGION Network 10: step 6: save received data 40002
   RUNG wire#powerrail
      { S7_Templates := "SrcType := USInt" } EQ_Contact(in1 := "dbTags_master_MPP04_2"."step", in2 := 6)
      Contact( "dbTags_master_MPP04_2".modbusMaster.done )
      wire#w1
      { S7_GenerateENO := "TRUE" } Move(in := "dbMasterData".data6_Licznik_objętość_VR_Adres_4.data[0], out1 => "dbModbusRTU_Reg".received_6_Licznik_objętość_VR_Adres_4.data[1])
      { S7_GenerateENO := "TRUE" } Move(in := "dbMasterData".data6_Licznik_objętość_VR_Adres_4.data[1], out1 => "dbModbusRTU_Reg".received_6_Licznik_objętość_VR_Adres_4.data[0])
      R_Coil( "dbTags_master_MPP04_2".modbusMaster.req )
   END_RUNG
   RUNG wire#w1
      { S7_GenerateENO := "TRUE" } Move(in := 7, out1 => "dbTags_master_MPP04_2"."step")
   END_RUNG
   // the same network as SCL:
   // ENO of a box is taken as its EN; it also drops when the box reports an error
   IF ("dbTags_master_MPP04_2"."step" = 6) AND "dbTags_master_MPP04_2".modbusMaster.done THEN
       "dbModbusRTU_Reg".received_6_Licznik_objętość_VR_Adres_4.data[1] := "dbMasterData".data6_Licznik_objętość_VR_Adres_4.data[0];
       "dbModbusRTU_Reg".received_6_Licznik_objętość_VR_Adres_4.data[0] := "dbMasterData".data6_Licznik_objętość_VR_Adres_4.data[1];
       "dbTags_master_MPP04_2".modbusMaster.req := FALSE;
       "dbTags_master_MPP04_2"."step" := 7;
   END_IF;
END_REGION

REGION Network 11: MODBUS RTU adress 27******step 9: read from slave 400011
   // Pobieramy Temperaturę w KN2
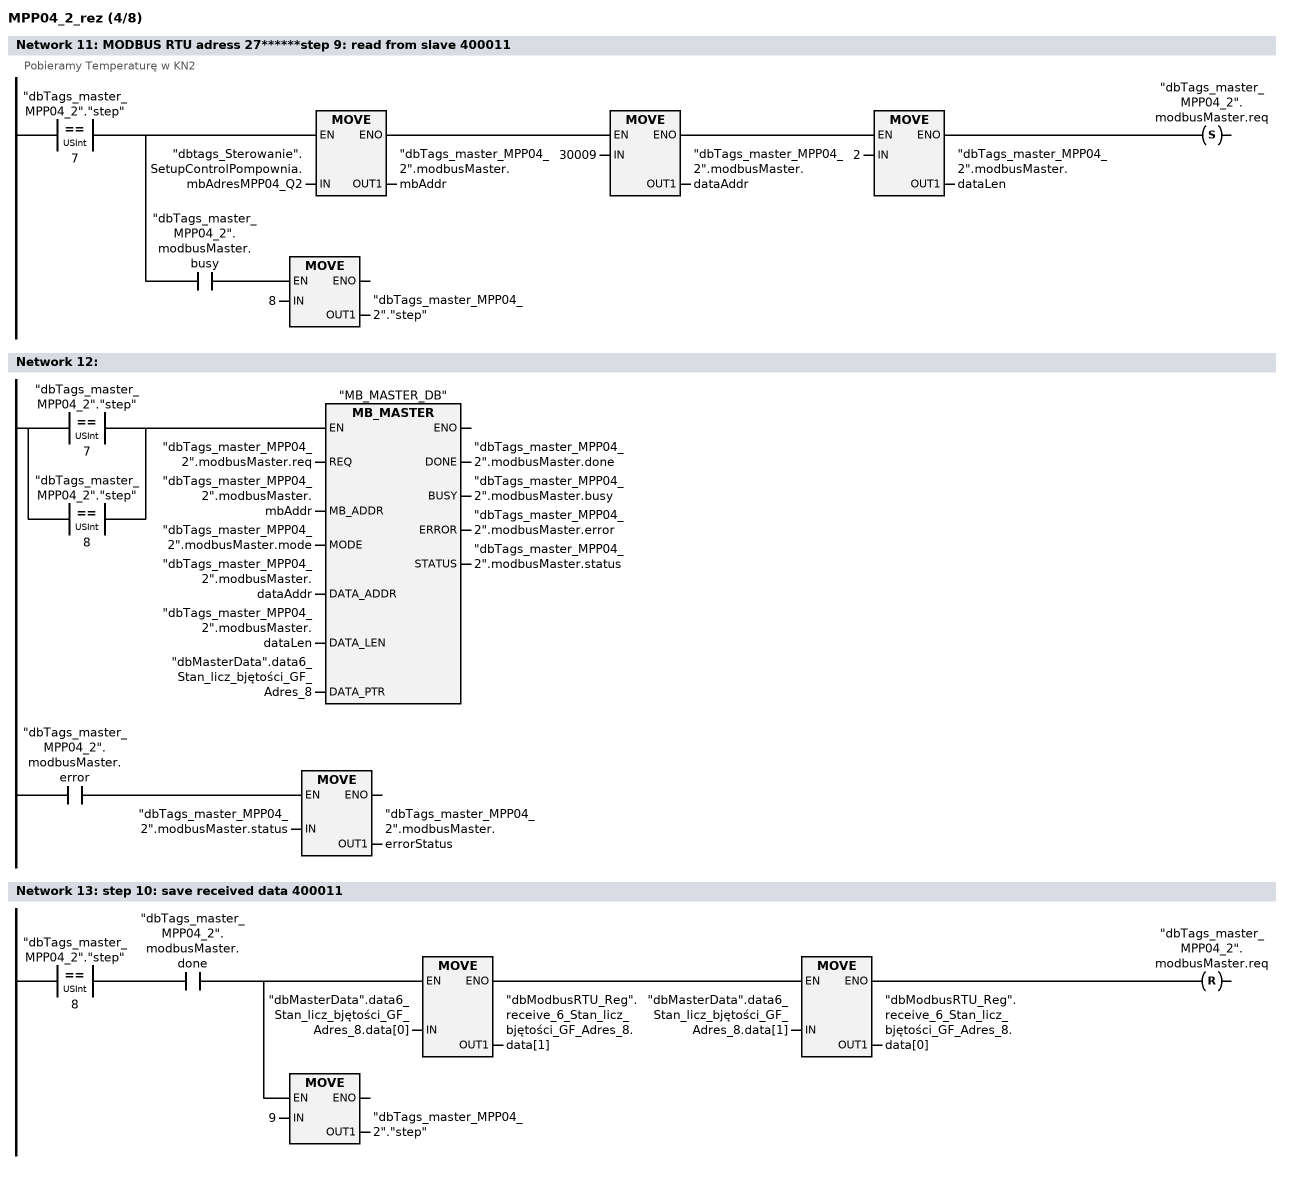
   RUNG wire#powerrail
      { S7_Templates := "SrcType := USInt" } EQ_Contact(in1 := "dbTags_master_MPP04_2"."step", in2 := 7)
      wire#w1
      Move(in := "dbtags_Sterowanie".SetupControlPompownia.mbAdresMPP04_Q2, out1 => "dbTags_master_MPP04_2".modbusMaster.mbAddr)
      { S7_GenerateENO := "TRUE" } Move(in := 30009, out1 => "dbTags_master_MPP04_2".modbusMaster.dataAddr)
      Move(in := 2, out1 => "dbTags_master_MPP04_2".modbusMaster.dataLen)
      S_Coil( "dbTags_master_MPP04_2".modbusMaster.req )
   END_RUNG
   RUNG wire#w1
      Contact( "dbTags_master_MPP04_2".modbusMaster.busy )
      { S7_GenerateENO := "TRUE" } Move(in := 8, out1 => "dbTags_master_MPP04_2"."step")
   END_RUNG
   // the same network as SCL:
   // ENO of a box is taken as its EN; it also drops when the box reports an error
   #_w1 := "dbTags_master_MPP04_2"."step" = 7;
   IF #_w1 THEN
       "dbTags_master_MPP04_2".modbusMaster.mbAddr := "dbtags_Sterowanie".SetupControlPompownia.mbAdresMPP04_Q2;
       "dbTags_master_MPP04_2".modbusMaster.dataAddr := 30009;
       "dbTags_master_MPP04_2".modbusMaster.dataLen := 2;
       "dbTags_master_MPP04_2".modbusMaster.req := TRUE;
   END_IF;
   IF #_w1 AND "dbTags_master_MPP04_2".modbusMaster.busy THEN "dbTags_master_MPP04_2"."step" := 8; END_IF;
END_REGION

REGION Network 12
   RUNG wire#powerrail
      { S7_Templates := "SrcType := USInt" } EQ_Contact(in1 := "dbTags_master_MPP04_2"."step", in2 := 7)
      wire#w1
      "MB_MASTER_DB".MB_MASTER(REQ := "dbTags_master_MPP04_2".modbusMaster.req, MB_ADDR := "dbTags_master_MPP04_2".modbusMaster.mbAddr, MODE := "dbTags_master_MPP04_2".modbusMaster.mode, DATA_ADDR := "dbTags_master_MPP04_2".modbusMaster.dataAddr, DATA_LEN := "dbTags_master_MPP04_2".modbusMaster.dataLen, DATA_PTR := "dbMasterData".data6_Stan_licz_bjętości_GF_Adres_8, DONE => "dbTags_master_MPP04_2".modbusMaster.done, BUSY => "dbTags_master_MPP04_2".modbusMaster.busy, ERROR => "dbTags_master_MPP04_2".modbusMaster.error, STATUS => "dbTags_master_MPP04_2".modbusMaster.status)
   END_RUNG
   RUNG wire#powerrail
      { S7_Templates := "SrcType := USInt" } EQ_Contact(in1 := "dbTags_master_MPP04_2"."step", in2 := 8)
   END_RUNG wire#w1
   RUNG wire#powerrail
      Contact( "dbTags_master_MPP04_2".modbusMaster.error )
      { S7_GenerateENO := "TRUE" } Move(in := "dbTags_master_MPP04_2".modbusMaster.status, out1 => "dbTags_master_MPP04_2".modbusMaster.errorStatus)
   END_RUNG
   // the same network as SCL:
   IF ("dbTags_master_MPP04_2"."step" = 7) OR ("dbTags_master_MPP04_2"."step" = 8) THEN
       "MB_MASTER_DB"(REQ := "dbTags_master_MPP04_2".modbusMaster.req,   // MB_MASTER
                      MB_ADDR := "dbTags_master_MPP04_2".modbusMaster.mbAddr,
                      MODE := "dbTags_master_MPP04_2".modbusMaster.mode,
                      DATA_ADDR := "dbTags_master_MPP04_2".modbusMaster.dataAddr,
                      DATA_LEN := "dbTags_master_MPP04_2".modbusMaster.dataLen,
                      DATA_PTR := "dbMasterData".data6_Stan_licz_bjętości_GF_Adres_8,
                      DONE => "dbTags_master_MPP04_2".modbusMaster.done,
                      BUSY => "dbTags_master_MPP04_2".modbusMaster.busy,
                      ERROR => "dbTags_master_MPP04_2".modbusMaster.error,
                      STATUS => "dbTags_master_MPP04_2".modbusMaster.status);
   END_IF;
   IF "dbTags_master_MPP04_2".modbusMaster.error THEN
       "dbTags_master_MPP04_2".modbusMaster.errorStatus := "dbTags_master_MPP04_2".modbusMaster.status;
   END_IF;
END_REGION

REGION Network 13: step 10: save received data 400011
   RUNG wire#powerrail
      { S7_Templates := "SrcType := USInt" } EQ_Contact(in1 := "dbTags_master_MPP04_2"."step", in2 := 8)
      Contact( "dbTags_master_MPP04_2".modbusMaster.done )
      wire#w1
      { S7_GenerateENO := "TRUE" } Move(in := "dbMasterData".data6_Stan_licz_bjętości_GF_Adres_8.data[0], out1 => "dbModbusRTU_Reg".receive_6_Stan_licz_bjętości_GF_Adres_8.data[1])
      { S7_GenerateENO := "TRUE" } Move(in := "dbMasterData".data6_Stan_licz_bjętości_GF_Adres_8.data[1], out1 => "dbModbusRTU_Reg".receive_6_Stan_licz_bjętości_GF_Adres_8.data[0])
      R_Coil( "dbTags_master_MPP04_2".modbusMaster.req )
   END_RUNG
   RUNG wire#w1
      { S7_GenerateENO := "TRUE" } Move(in := 9, out1 => "dbTags_master_MPP04_2"."step")
   END_RUNG
   // the same network as SCL:
   // ENO of a box is taken as its EN; it also drops when the box reports an error
   IF ("dbTags_master_MPP04_2"."step" = 8) AND "dbTags_master_MPP04_2".modbusMaster.done THEN
       "dbModbusRTU_Reg".receive_6_Stan_licz_bjętości_GF_Adres_8.data[1] := "dbMasterData".data6_Stan_licz_bjętości_GF_Adres_8.data[0];
       "dbModbusRTU_Reg".receive_6_Stan_licz_bjętości_GF_Adres_8.data[0] := "dbMasterData".data6_Stan_licz_bjętości_GF_Adres_8.data[1];
       "dbTags_master_MPP04_2".modbusMaster.req := FALSE;
       "dbTags_master_MPP04_2"."step" := 9;
   END_IF;
END_REGION

REGION Network 14: MODBUS RTU adress 27******step 11: read from slave 40007
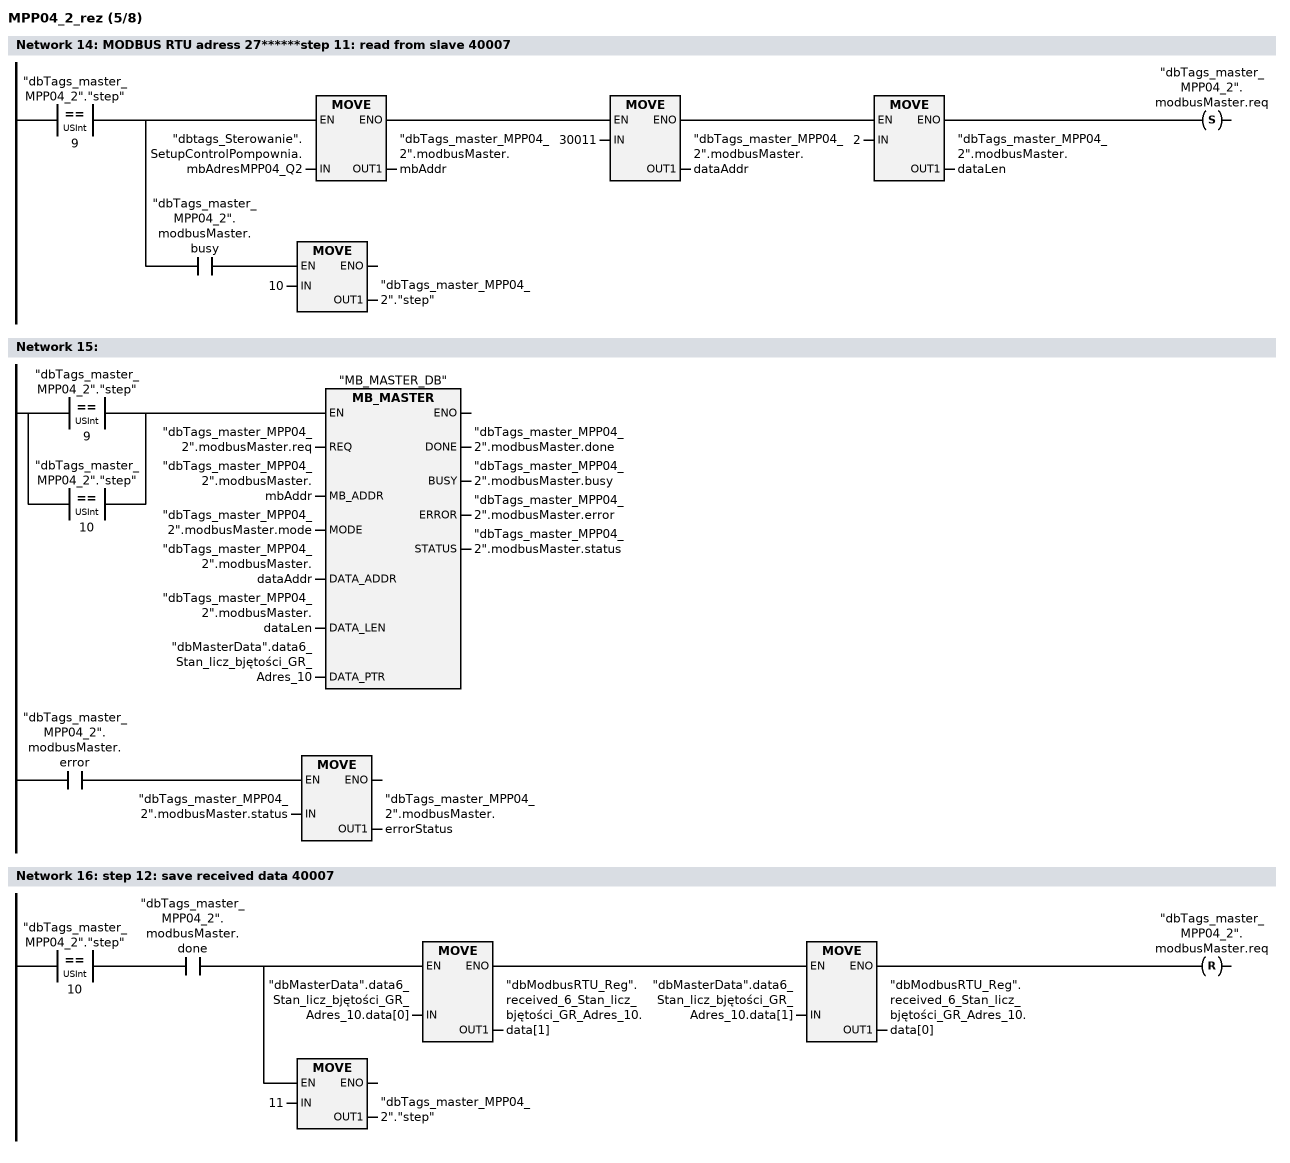
   RUNG wire#powerrail
      { S7_Templates := "SrcType := USInt" } EQ_Contact(in1 := "dbTags_master_MPP04_2"."step", in2 := 9)
      wire#w1
      Move(in := "dbtags_Sterowanie".SetupControlPompownia.mbAdresMPP04_Q2, out1 => "dbTags_master_MPP04_2".modbusMaster.mbAddr)
      { S7_GenerateENO := "TRUE" } Move(in := 30011, out1 => "dbTags_master_MPP04_2".modbusMaster.dataAddr)
      Move(in := 2, out1 => "dbTags_master_MPP04_2".modbusMaster.dataLen)
      S_Coil( "dbTags_master_MPP04_2".modbusMaster.req )
   END_RUNG
   RUNG wire#w1
      Contact( "dbTags_master_MPP04_2".modbusMaster.busy )
      { S7_GenerateENO := "TRUE" } Move(in := 10, out1 => "dbTags_master_MPP04_2"."step")
   END_RUNG
   // the same network as SCL:
   // ENO of a box is taken as its EN; it also drops when the box reports an error
   #_w1 := "dbTags_master_MPP04_2"."step" = 9;
   IF #_w1 THEN
       "dbTags_master_MPP04_2".modbusMaster.mbAddr := "dbtags_Sterowanie".SetupControlPompownia.mbAdresMPP04_Q2;
       "dbTags_master_MPP04_2".modbusMaster.dataAddr := 30011;
       "dbTags_master_MPP04_2".modbusMaster.dataLen := 2;
       "dbTags_master_MPP04_2".modbusMaster.req := TRUE;
   END_IF;
   IF #_w1 AND "dbTags_master_MPP04_2".modbusMaster.busy THEN "dbTags_master_MPP04_2"."step" := 10; END_IF;
END_REGION

REGION Network 15
   RUNG wire#powerrail
      { S7_Templates := "SrcType := USInt" } EQ_Contact(in1 := "dbTags_master_MPP04_2"."step", in2 := 9)
      wire#w1
      "MB_MASTER_DB".MB_MASTER(REQ := "dbTags_master_MPP04_2".modbusMaster.req, MB_ADDR := "dbTags_master_MPP04_2".modbusMaster.mbAddr, MODE := "dbTags_master_MPP04_2".modbusMaster.mode, DATA_ADDR := "dbTags_master_MPP04_2".modbusMaster.dataAddr, DATA_LEN := "dbTags_master_MPP04_2".modbusMaster.dataLen, DATA_PTR := "dbMasterData".data6_Stan_licz_bjętości_GR_Adres_10, DONE => "dbTags_master_MPP04_2".modbusMaster.done, BUSY => "dbTags_master_MPP04_2".modbusMaster.busy, ERROR => "dbTags_master_MPP04_2".modbusMaster.error, STATUS => "dbTags_master_MPP04_2".modbusMaster.status)
   END_RUNG
   RUNG wire#powerrail
      { S7_Templates := "SrcType := USInt" } EQ_Contact(in1 := "dbTags_master_MPP04_2"."step", in2 := 10)
   END_RUNG wire#w1
   RUNG wire#powerrail
      Contact( "dbTags_master_MPP04_2".modbusMaster.error )
      { S7_GenerateENO := "TRUE" } Move(in := "dbTags_master_MPP04_2".modbusMaster.status, out1 => "dbTags_master_MPP04_2".modbusMaster.errorStatus)
   END_RUNG
   // the same network as SCL:
   IF ("dbTags_master_MPP04_2"."step" = 9) OR ("dbTags_master_MPP04_2"."step" = 10) THEN
       "MB_MASTER_DB"(REQ := "dbTags_master_MPP04_2".modbusMaster.req,   // MB_MASTER
                      MB_ADDR := "dbTags_master_MPP04_2".modbusMaster.mbAddr,
                      MODE := "dbTags_master_MPP04_2".modbusMaster.mode,
                      DATA_ADDR := "dbTags_master_MPP04_2".modbusMaster.dataAddr,
                      DATA_LEN := "dbTags_master_MPP04_2".modbusMaster.dataLen,
                      DATA_PTR := "dbMasterData".data6_Stan_licz_bjętości_GR_Adres_10,
                      DONE => "dbTags_master_MPP04_2".modbusMaster.done,
                      BUSY => "dbTags_master_MPP04_2".modbusMaster.busy,
                      ERROR => "dbTags_master_MPP04_2".modbusMaster.error,
                      STATUS => "dbTags_master_MPP04_2".modbusMaster.status);
   END_IF;
   IF "dbTags_master_MPP04_2".modbusMaster.error THEN
       "dbTags_master_MPP04_2".modbusMaster.errorStatus := "dbTags_master_MPP04_2".modbusMaster.status;
   END_IF;
END_REGION

REGION Network 16: step 12: save received data 40007
   RUNG wire#powerrail
      { S7_Templates := "SrcType := USInt" } EQ_Contact(in1 := "dbTags_master_MPP04_2"."step", in2 := 10)
      Contact( "dbTags_master_MPP04_2".modbusMaster.done )
      wire#w1
      { S7_GenerateENO := "TRUE" } Move(in := "dbMasterData".data6_Stan_licz_bjętości_GR_Adres_10.data[0], out1 => "dbModbusRTU_Reg".received_6_Stan_licz_bjętości_GR_Adres_10.data[1])
      { S7_GenerateENO := "TRUE" } Move(in := "dbMasterData".data6_Stan_licz_bjętości_GR_Adres_10.data[1], out1 => "dbModbusRTU_Reg".received_6_Stan_licz_bjętości_GR_Adres_10.data[0])
      R_Coil( "dbTags_master_MPP04_2".modbusMaster.req )
   END_RUNG
   RUNG wire#w1
      { S7_GenerateENO := "TRUE" } Move(in := 11, out1 => "dbTags_master_MPP04_2"."step")
   END_RUNG
   // the same network as SCL:
   // ENO of a box is taken as its EN; it also drops when the box reports an error
   IF ("dbTags_master_MPP04_2"."step" = 10) AND "dbTags_master_MPP04_2".modbusMaster.done THEN
       "dbModbusRTU_Reg".received_6_Stan_licz_bjętości_GR_Adres_10.data[1] := "dbMasterData".data6_Stan_licz_bjętości_GR_Adres_10.data[0];
       "dbModbusRTU_Reg".received_6_Stan_licz_bjętości_GR_Adres_10.data[0] := "dbMasterData".data6_Stan_licz_bjętości_GR_Adres_10.data[1];
       "dbTags_master_MPP04_2".modbusMaster.req := FALSE;
       "dbTags_master_MPP04_2"."step" := 11;
   END_IF;
END_REGION

REGION Network 17: MODBUS RTU adress 27******step 15: read from slave 40009
   // Pobieramy  status urządzenia
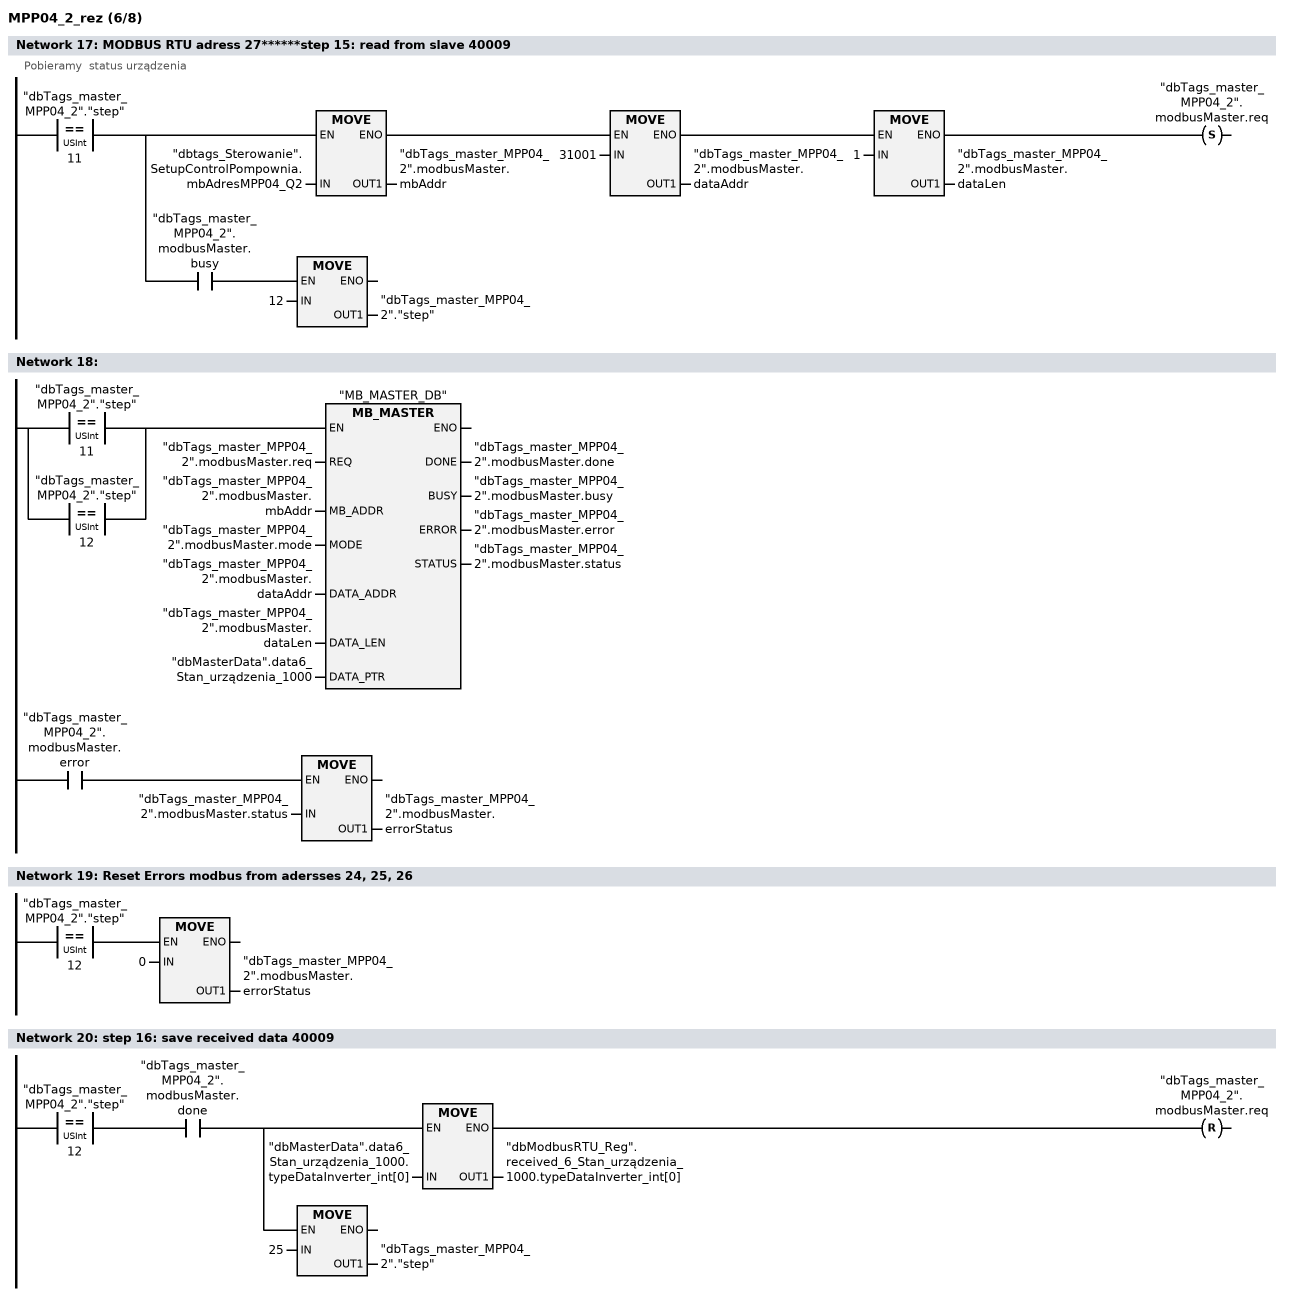
   RUNG wire#powerrail
      { S7_Templates := "SrcType := USInt" } EQ_Contact(in1 := "dbTags_master_MPP04_2"."step", in2 := 11)
      wire#w1
      Move(in := "dbtags_Sterowanie".SetupControlPompownia.mbAdresMPP04_Q2, out1 => "dbTags_master_MPP04_2".modbusMaster.mbAddr)
      { S7_GenerateENO := "TRUE" } Move(in := 31001, out1 => "dbTags_master_MPP04_2".modbusMaster.dataAddr)
      Move(in := 1, out1 => "dbTags_master_MPP04_2".modbusMaster.dataLen)
      S_Coil( "dbTags_master_MPP04_2".modbusMaster.req )
   END_RUNG
   RUNG wire#w1
      Contact( "dbTags_master_MPP04_2".modbusMaster.busy )
      { S7_GenerateENO := "TRUE" } Move(in := 12, out1 => "dbTags_master_MPP04_2"."step")
   END_RUNG
   // the same network as SCL:
   // ENO of a box is taken as its EN; it also drops when the box reports an error
   #_w1 := "dbTags_master_MPP04_2"."step" = 11;
   IF #_w1 THEN
       "dbTags_master_MPP04_2".modbusMaster.mbAddr := "dbtags_Sterowanie".SetupControlPompownia.mbAdresMPP04_Q2;
       "dbTags_master_MPP04_2".modbusMaster.dataAddr := 31001;
       "dbTags_master_MPP04_2".modbusMaster.dataLen := 1;
       "dbTags_master_MPP04_2".modbusMaster.req := TRUE;
   END_IF;
   IF #_w1 AND "dbTags_master_MPP04_2".modbusMaster.busy THEN "dbTags_master_MPP04_2"."step" := 12; END_IF;
END_REGION

REGION Network 18
   RUNG wire#powerrail
      { S7_Templates := "SrcType := USInt" } EQ_Contact(in1 := "dbTags_master_MPP04_2"."step", in2 := 11)
      wire#w1
      "MB_MASTER_DB".MB_MASTER(REQ := "dbTags_master_MPP04_2".modbusMaster.req, MB_ADDR := "dbTags_master_MPP04_2".modbusMaster.mbAddr, MODE := "dbTags_master_MPP04_2".modbusMaster.mode, DATA_ADDR := "dbTags_master_MPP04_2".modbusMaster.dataAddr, DATA_LEN := "dbTags_master_MPP04_2".modbusMaster.dataLen, DATA_PTR := "dbMasterData".data6_Stan_urządzenia_1000, DONE => "dbTags_master_MPP04_2".modbusMaster.done, BUSY => "dbTags_master_MPP04_2".modbusMaster.busy, ERROR => "dbTags_master_MPP04_2".modbusMaster.error, STATUS => "dbTags_master_MPP04_2".modbusMaster.status)
   END_RUNG
   RUNG wire#powerrail
      { S7_Templates := "SrcType := USInt" } EQ_Contact(in1 := "dbTags_master_MPP04_2"."step", in2 := 12)
   END_RUNG wire#w1
   RUNG wire#powerrail
      Contact( "dbTags_master_MPP04_2".modbusMaster.error )
      { S7_GenerateENO := "TRUE" } Move(in := "dbTags_master_MPP04_2".modbusMaster.status, out1 => "dbTags_master_MPP04_2".modbusMaster.errorStatus)
   END_RUNG
   // the same network as SCL:
   IF ("dbTags_master_MPP04_2"."step" = 11) OR ("dbTags_master_MPP04_2"."step" = 12) THEN
       "MB_MASTER_DB"(REQ := "dbTags_master_MPP04_2".modbusMaster.req,   // MB_MASTER
                      MB_ADDR := "dbTags_master_MPP04_2".modbusMaster.mbAddr,
                      MODE := "dbTags_master_MPP04_2".modbusMaster.mode,
                      DATA_ADDR := "dbTags_master_MPP04_2".modbusMaster.dataAddr,
                      DATA_LEN := "dbTags_master_MPP04_2".modbusMaster.dataLen,
                      DATA_PTR := "dbMasterData".data6_Stan_urządzenia_1000,
                      DONE => "dbTags_master_MPP04_2".modbusMaster.done,
                      BUSY => "dbTags_master_MPP04_2".modbusMaster.busy,
                      ERROR => "dbTags_master_MPP04_2".modbusMaster.error,
                      STATUS => "dbTags_master_MPP04_2".modbusMaster.status);
   END_IF;
   IF "dbTags_master_MPP04_2".modbusMaster.error THEN
       "dbTags_master_MPP04_2".modbusMaster.errorStatus := "dbTags_master_MPP04_2".modbusMaster.status;
   END_IF;
END_REGION

REGION Network 19: Reset Errors modbus from adersses 24, 25, 26
   RUNG wire#powerrail
      { S7_Templates := "SrcType := USInt" } EQ_Contact(in1 := "dbTags_master_MPP04_2"."step", in2 := 12)
      { S7_GenerateENO := "TRUE" } Move(in := 0, out1 => "dbTags_master_MPP04_2".modbusMaster.errorStatus)
   END_RUNG
   // the same network as SCL:
   IF "dbTags_master_MPP04_2"."step" = 12 THEN "dbTags_master_MPP04_2".modbusMaster.errorStatus := 0; END_IF;
END_REGION

REGION Network 20: step 16: save received data 40009
   RUNG wire#powerrail
      { S7_Templates := "SrcType := USInt" } EQ_Contact(in1 := "dbTags_master_MPP04_2"."step", in2 := 12)
      Contact( "dbTags_master_MPP04_2".modbusMaster.done )
      wire#w1
      { S7_GenerateENO := "TRUE" } Move(in := "dbMasterData".data6_Stan_urządzenia_1000.typeDataInverter_int[0], out1 => "dbModbusRTU_Reg".received_6_Stan_urządzenia_1000.typeDataInverter_int[0])
      R_Coil( "dbTags_master_MPP04_2".modbusMaster.req )
   END_RUNG
   RUNG wire#w1
      { S7_GenerateENO := "TRUE" } Move(in := 25, out1 => "dbTags_master_MPP04_2"."step")
   END_RUNG
   // the same network as SCL:
   // ENO of a box is taken as its EN; it also drops when the box reports an error
   IF ("dbTags_master_MPP04_2"."step" = 12) AND "dbTags_master_MPP04_2".modbusMaster.done THEN
       "dbModbusRTU_Reg".received_6_Stan_urządzenia_1000.typeDataInverter_int[0] := "dbMasterData".data6_Stan_urządzenia_1000.typeDataInverter_int[0];
       "dbTags_master_MPP04_2".modbusMaster.req := FALSE;
       "dbTags_master_MPP04_2"."step" := 25;
   END_IF;
END_REGION

REGION Network 21: Znacznik błedu komunikacji modbus
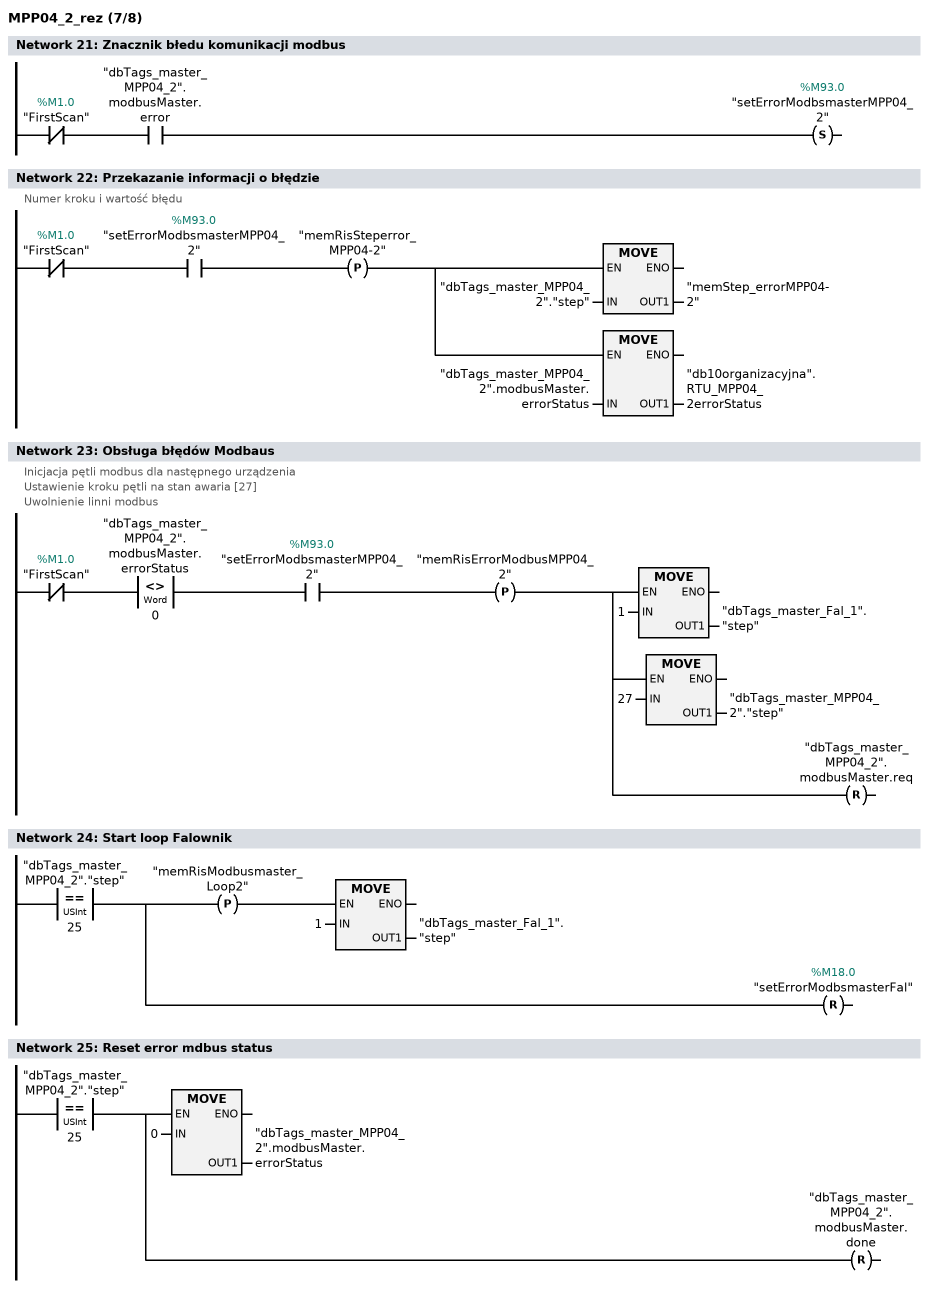
   RUNG wire#powerrail
      I_Contact( "FirstScan" )
      Contact( "dbTags_master_MPP04_2".modbusMaster.error )
      S_Coil( "setErrorModbsmasterMPP04_2" )
   END_RUNG
   // the same network as SCL:
   IF NOT "FirstScan" AND "dbTags_master_MPP04_2".modbusMaster.error THEN
       "setErrorModbsmasterMPP04_2" := TRUE;
   END_IF;
END_REGION

REGION Network 22: Przekazanie informacji o błędzie
   // Numer kroku i wartość błędu
   RUNG wire#powerrail
      I_Contact( "FirstScan" )
      Contact( "setErrorModbsmasterMPP04_2" )
      P_Trig( "memRisSteperror_MPP04-2" )
      wire#w1
      Move(in := "dbTags_master_MPP04_2"."step", out1 => "memStep_errorMPP04-2")
   END_RUNG
   RUNG wire#w1
      { S7_GenerateENO := "TRUE" } Move(in := "dbTags_master_MPP04_2".modbusMaster.errorStatus, out1 => "db10organizacyjna".RTU_MPP04_2errorStatus)
   END_RUNG
   // the same network as SCL:
   #_w1 := NOT "FirstScan" AND "setErrorModbsmasterMPP04_2";
   #_w2 := #_w1 AND NOT "memRisSteperror_MPP04-2";   // rising edge
   "memRisSteperror_MPP04-2" := #_w1;
   IF #_w2 THEN
       "memStep_errorMPP04-2" := "dbTags_master_MPP04_2"."step";
       "db10organizacyjna".RTU_MPP04_2errorStatus := "dbTags_master_MPP04_2".modbusMaster.errorStatus;
   END_IF;
END_REGION

REGION Network 23: Obsługa błędów Modbaus
   // Inicjacja pętli modbus dla następnego urządzenia
   // Ustawienie kroku pętli na stan awaria [27]
   // Uwolnienie linni modbus
   RUNG wire#powerrail
      I_Contact( "FirstScan" )
      { S7_Templates := "SrcType := Word" } NE_Contact(in1 := "dbTags_master_MPP04_2".modbusMaster.errorStatus, in2 := 0)
      Contact( "setErrorModbsmasterMPP04_2" )
      P_Trig( "memRisErrorModbusMPP04_2" )
      wire#w1
      { S7_GenerateENO := "TRUE" } Move(in := 1, out1 => "dbTags_master_Fal_1"."step")
   END_RUNG
   RUNG wire#w1
      { S7_GenerateENO := "TRUE" } Move(in := 27, out1 => "dbTags_master_MPP04_2"."step")
   END_RUNG
   RUNG wire#w1
      R_Coil( "dbTags_master_MPP04_2".modbusMaster.req )
   END_RUNG
   // the same network as SCL:
   #_w1 := NOT "FirstScan" AND ("dbTags_master_MPP04_2".modbusMaster.errorStatus <> 0) AND "setErrorModbsmasterMPP04_2";
   #_w2 := #_w1 AND NOT "memRisErrorModbusMPP04_2";   // rising edge
   "memRisErrorModbusMPP04_2" := #_w1;
   IF #_w2 THEN
       "dbTags_master_Fal_1"."step" := 1;
       "dbTags_master_MPP04_2"."step" := 27;
       "dbTags_master_MPP04_2".modbusMaster.req := FALSE;
   END_IF;
END_REGION

REGION Network 24: Start loop Falownik
   RUNG wire#powerrail
      { S7_Templates := "SrcType := USInt" } EQ_Contact(in1 := "dbTags_master_MPP04_2"."step", in2 := 25)
      wire#w1
      P_Trig( "memRisModbusmaster_Loop2" )
      { S7_GenerateENO := "TRUE" } Move(in := 1, out1 => "dbTags_master_Fal_1"."step")
   END_RUNG
   RUNG wire#w1
      R_Coil( "setErrorModbsmasterFal" )
   END_RUNG
   // the same network as SCL:
   #_w1 := "dbTags_master_MPP04_2"."step" = 25;
   #_w2 := #_w1 AND NOT "memRisModbusmaster_Loop2";   // rising edge
   "memRisModbusmaster_Loop2" := #_w1;
   IF #_w2 THEN "dbTags_master_Fal_1"."step" := 1; END_IF;
   IF #_w1 THEN "setErrorModbsmasterFal" := FALSE; END_IF;
END_REGION

REGION Network 25: Reset error mdbus status
   RUNG wire#powerrail
      { S7_Templates := "SrcType := USInt" } EQ_Contact(in1 := "dbTags_master_MPP04_2"."step", in2 := 25)
      wire#w1
      { S7_GenerateENO := "TRUE" } Move(in := 0, out1 => "dbTags_master_MPP04_2".modbusMaster.errorStatus)
   END_RUNG
   RUNG wire#w1
      R_Coil( "dbTags_master_MPP04_2".modbusMaster.done )
   END_RUNG
   // the same network as SCL:
   IF "dbTags_master_MPP04_2"."step" = 25 THEN
       "dbTags_master_MPP04_2".modbusMaster.errorStatus := 0;
       "dbTags_master_MPP04_2".modbusMaster.done := FALSE;
   END_IF;
END_REGION

REGION Network 26: Reset Znacznik błedu komunikacji modbus
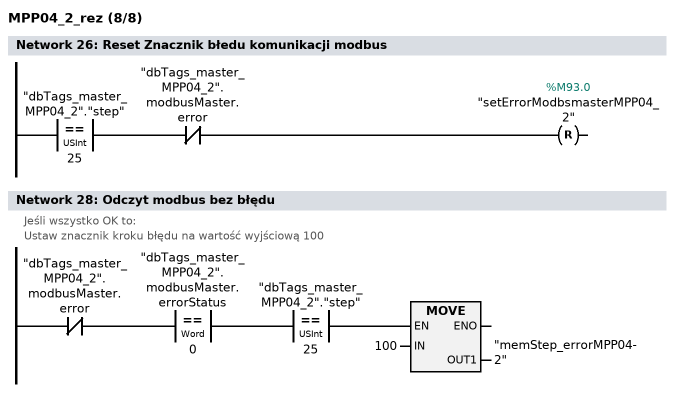
   RUNG wire#powerrail
      { S7_Templates := "SrcType := USInt" } EQ_Contact(in1 := "dbTags_master_MPP04_2"."step", in2 := 25)
      I_Contact( "dbTags_master_MPP04_2".modbusMaster.error )
      R_Coil( "setErrorModbsmasterMPP04_2" )
   END_RUNG
   // the same network as SCL:
   IF ("dbTags_master_MPP04_2"."step" = 25) AND NOT "dbTags_master_MPP04_2".modbusMaster.error THEN
       "setErrorModbsmasterMPP04_2" := FALSE;
   END_IF;
END_REGION

REGION Network 28: Odczyt modbus bez błędu
   // Jeśli wszystko OK to:
   // Ustaw znacznik kroku błędu na wartość wyjściową 100
   RUNG wire#powerrail
      I_Contact( "dbTags_master_MPP04_2".modbusMaster.error )
      { S7_Templates := "SrcType := Word" } EQ_Contact(in1 := "dbTags_master_MPP04_2".modbusMaster.errorStatus, in2 := 0)
      { S7_Templates := "SrcType := USInt" } EQ_Contact(in1 := "dbTags_master_MPP04_2"."step", in2 := 25)
      { S7_GenerateENO := "TRUE" } Move(in := 100, out1 => "memStep_errorMPP04-2")
   END_RUNG
   // the same network as SCL:
   IF NOT "dbTags_master_MPP04_2".modbusMaster.error AND ("dbTags_master_MPP04_2".modbusMaster.errorStatus = 0) AND ("dbTags_master_MPP04_2"."step" = 25) THEN
       "memStep_errorMPP04-2" := 100;
   END_IF;
END_REGION
END_FUNCTION

ORGANIZATION_BLOCK "Cyclic interrupt_1"
{ S7_Optimized_Access := 'TRUE' }
VERSION : 0.1

BEGIN
	(*
	//=============================================================================
	//(JZWiK S.A Radosław Tecmer)
	//(c)Copyright (2021) All Rights Reserved
	//-----------------------------------------------------------------------------
	//Testowane z:   (system docelowy z  FW 4.4)
	//Pakiet inżynierski:   TIA Portal (V14 Sp1 Update 9)
	//Ograniczenia:  ( - )
	//Wymagania:  (minimalne S7-1200 CPU 1215C FW 4.2 .)
	//Funkcjonalnośc: (Pobranie wartości z wejść analogowych )
	//-----------------------------------------------------------------------------
	//Zmainy wprowadzone:
	//Wersja  Data       Osoba wprowadzająca zmiany - ekspert
	//01.00.00 11.01.2022 (Tecmer Radosław - twórca) Pieresza wersja 01.00.00
	//=============================================================================
	*)
	// Analogi 
	// ciśnienie przetłaczania miasto 
	"dbdane".PV_analaog_B6 := "IW64":P;
	// ciśnienie pompownia
	"dbdane".PV_analaog_B7 := "IW66":P;
	//ciśnienie ssania
	"dbdane".PV_analaog_B8 := "IW68":P;
	
	
END_ORGANIZATION_BLOCK

FUNCTION "Zmienne_dbModbusMaster_1" : Void
{ S7_Optimized_Access := 'TRUE' }
AUTHOR : RTecmer
FAMILY : 'HMI(XM)'
VERSION : 0.1
//Przekazywanie zmiennych między urządzeniami

BEGIN
	(*
	//=============================================================================
	//(JZWiK S.A Radosław Tecmer)
	//(c)Copyright (2021) All Rights Reserved
	//-----------------------------------------------------------------------------
	//Testowane z:   (system docelowy z  FW 4.2)
	//Pakiet inżynierski:   TIA Portal (V14 Sp1 Update 9)
	//Ograniczenia:  ( - )
	//Wymagania:  (minimalne S7-1200 CPU 1214 FW 3.2 .)
	//Funkcjonalnośc: (Kopiowanie bloków danych między blokiem danych Modbus -SCADA  )
	//-----------------------------------------------------------------------------
	//Zmainy wprowadzone:
	//Wersja  Data       Osoba wprowadzająca zmiany - ekspert
	//01.00.00 17.11.2021 (Tecmer Radosław - twórca) Pieresza wersja 01.00.00
	//=============================================================================
	*)
	
	REGION Analogi
	  // 
	
	  
	  
	END_REGION
	
	
	
	
	
	 
	
	
	
	
	
	
	
	
	
	
	
	
	
	
	
	
	
	
	
	
	
	
END_FUNCTION

FUNCTION "Block_1" : Void
{ S7_Optimized_Access := 'TRUE' }
VERSION : 0.1

BEGIN
	
	
	//
	
	IF "dbTimersForDrivers".Timer_OFF_Inverter_P1.Q OR "dbTimersForDrivers".Timer_OFF_Inverter_P2.Q OR
	  "dbTimersForDrivers".Timer_OFF_Inverter_P3.Q OR "dbTimersForDrivers".Timer_OFF_Inverter_P4.Q
	  
	THEN
	  "IsModeAut" := TRUE;
	  
	  IF "bitH_Aut_Man_P1" THEN
	    // Statement section IF
	    %DB100.DBX0.7 := TRUE;
	    %DB100.DBX1.7 := TRUE;
	    ;
	  END_IF;
	  IF "bitH_Aut_Man_P2" THEN
	    // Statement section IF
	    %DB100.DBX2.7 := TRUE;
	    %DB100.DBX3.7 := TRUE;
	    ;
	  END_IF;
	  IF "bitH_Aut_Man_P3" THEN
	    // Statement section IF
	    %DB100.DBX4.7 := TRUE;
	    %DB100.DBX5.7 := TRUE;
	    ;
	  END_IF;
	  IF "bitH_Aut_Man_P4" THEN
	    // Statement section IF
	    %DB100.DBX6.7 := TRUE;
	    %DB100.DBX7.7 := TRUE;
	    ;
	  END_IF;
	  
	END_IF;
	
	CASE "dbHold_RRG".set_res_bity_tryb_napędów_1 OF
	    //256:  // Ustawienie bitu Aut dla Drive Z1
	    //"dbHold_RRG".Sending.set_res_bity_tryb_napędów_1 := 256;
	    //;
	    //512:  // Ustawienie bitu Aut dla Drive Z2
	    //"dbHold_RRG".Sending.set_res_bity_tryb_napędów_1 := 512;
	    //;
	  1024:  // Ustawienie bitu Aut dla Drive Z3
	    "dbHold_RRG".Sending.set_res_bity_tryb_napędów_1 := 1024;
	    ;
	  2048:  //Ustawienie bitu Aut dla Drive Z4
	    "dbHold_RRG".Sending.set_res_bity_tryb_napędów_1 := 2048;
	    ;
	  4096:  //Ustawienie bitu Aut dla Drive Z5
	    "dbHold_RRG".Sending.set_res_bity_tryb_napędów_1 := 4096;
	    ;
	  8192:  //Ustawienie bitu Aut dla Drive Z6
	    "dbHold_RRG".Sending.set_res_bity_tryb_napędów_1 := 8192;
	    ;
	  16384:  //Ustawienie bitu Reset dla Drive Z7
	    "dbHold_RRG".Sending.set_res_bity_tryb_napędów_1 := 16384;
	    ;
	  32768:  //Ustawienie bitu Aut dla Drive Z8
	    "dbHold_RRG".Sending.set_res_bity_tryb_napędów_1 := 32768;
	    
	    
	    ;
	  ELSE  // Statement section ELSE
	    ;
	END_CASE;
	
	
	CASE "dbHold_RRG".set_res_bity_tryb_napędów_2 OF
	  1:  // Ustawienie bitu Aut dla Drive Z1
	    "dbHold_RRG".Sending.set_res_bity_tryb_napędów_2 := 1;
	    ;
	  2:  // Ustawienie bitu Aut dla Drive Z2
	    "dbHold_RRG".Sending.set_res_bity_tryb_napędów_2 := 2;
	    
	  4:  // Ustawienie bitu Aut dla Drive Z2
	    "dbHold_RRG".Sending.set_res_bity_tryb_napędów_2 := 4;
	    
	  8:  // Ustawienie bitu Aut dla Drive Z2
	    "dbHold_RRG".Sending.set_res_bity_tryb_napędów_2 := 8;
	    
	  16:  // Ustawienie bitu Aut dla Drive Z2
	    "dbHold_RRG".Sending.set_res_bity_tryb_napędów_2 := 16;
	    
	  32:  // Ustawienie bitu Aut dla Drive Z2
	    "dbHold_RRG".Sending.set_res_bity_tryb_napędów_2 := 32;
	    
	  64:  // Ustawienie bitu Aut dla Drive Z2
	    "dbHold_RRG".Sending.set_res_bity_tryb_napędów_2 := 64;
	    
	  128:  // Ustawienie bitu Aut dla Drive Z2
	    "dbHold_RRG".Sending.set_res_bity_tryb_napędów_2 := 128;
	    
	  256:  // Ustawienie bitu Aut dla Drive Z2
	    "dbHold_RRG".Sending.set_res_bity_tryb_napędów_2 := 256;
	    
	  512:  // Ustawienie bitu Aut dla Drive Z2
	    "dbHold_RRG".Sending.set_res_bity_tryb_napędów_2 := 512;
	    
	  1024:  // Ustawienie bitu Aut dla Drive Z2
	    "dbHold_RRG".Sending.set_res_bity_tryb_napędów_2 := 1024;
	    
	  2048:  // Ustawienie bitu Aut dla Drive Z2
	    "dbHold_RRG".Sending.set_res_bity_tryb_napędów_2 := 2048;
	    
	  4096:  // Ustawienie bitu Aut dla Drive Z2
	    "dbHold_RRG".Sending.set_res_bity_tryb_napędów_2 := 4096;
	    
	  8192:  // Ustawienie bitu Aut dla Drive Z2
	    "dbHold_RRG".Sending.set_res_bity_tryb_napędów_2 := 8192;
	    
	  16384:  // Ustawienie bitu Aut dla Drive Z2
	    "dbHold_RRG".Sending.set_res_bity_tryb_napędów_2 := 16384;
	    
	  32768:  // Ustawienie bitu Aut dla Drive Z2
	    "dbHold_RRG".Sending.set_res_bity_tryb_napędów_2 := 32768;
	    
	    
	    ;
	  ELSE  // Statement section ELSE
	    ;
	END_CASE;
	
	
	
	
END_FUNCTION

FUNCTION "Sterowanie awaryje barMax" : Void
TITLE = Processing of the currently set oxygen value
{ S7_Optimized_Access := 'TRUE' }
AUTHOR : rtecmer
VERSION : 0.1
//Funkcja wyznacza aktualne źródło zygnału zadawania wartości bar na podstawie wybranej obcji zbiornika sterującego.
   VAR_INPUT 
      Switch_model_control : Int;   // Wybór model sterowania
      Set_Miasto : Real;   // Zadana wartość cisnienia [bar] przetłaczanie
      Set_Magistrala : Real;   // Zadana wartość ciśnienia [bar] dosilanie
   END_VAR

   VAR_OUTPUT 
      posBar : Real;   // Przechwycona wartość bar
   END_VAR

   VAR_TEMP 
      tmpBar_control : Bool;   // Przełącznik kontroli źródła sygnału wartości zadanej
   END_VAR


BEGIN
	//Funkcja wyznacza aktualne źródło zygnału zadawania wartości bar na podstawie
	//wybranej obcji zbiornika sterującego.
	
	//
	#tmpBar_control := TRUE;
	
	REGION Przechwycenie zadanej wartości bar 
	  // ustalenie począdkowej wartości podczas stsrt redukcji
	  IF #tmpBar_control THEN
	    // Przechwycenia wartości zadanej bar 
	    CASE #Switch_model_control OF
	      0: // Wyłaczone
	        ;
	      1:  // Dosilanie magistrala
	        #posBar := #Set_Magistrala;
	      2:  // Zadany z komory 2
	        #posBar := #Set_Miasto;
	      3: // automat
	        ;
	      ELSE  // 
	        ;
	    END_CASE;
	  END_IF;
	  
	END_REGION
END_FUNCTION

FUNCTION "SclScaleLinearRealToInt" : Int
{ S7_Optimized_Access := 'TRUE' }
VERSION : 0.1
   VAR_INPUT 
      x : Real;
      yMin : Int;
      yMax : Int;
      x0 : Real;
      y0 : Int;
      x1 : Real;
      y1 : Int;
   END_VAR

   VAR_TEMP 
      tempY0real : Real;
      tempY1real : Real;
      tempYreal : Real;
      tempYminReal : Real;
      tempYmaxReal : Real;
   END_VAR


BEGIN
	#tempY0real := INT_TO_REAL(#y0);
	#tempY1real := INT_TO_REAL(#y1);
	#tempYminReal := INT_TO_REAL(#yMin);
	#tempYmaxReal := INT_TO_REAL(#yMax);
	
	IF (#y1 - #y0) = 0 OR (#x1 - #x0) = 0 OR (#x - #x0) = 0 OR #yMin > #yMax
	THEN
	    #SclScaleLinearRealToInt := 0;
	ELSE
	    #tempYreal := (#tempY1real - #tempY0real) / (#x1 - #x0) * (#x - #x0) + #tempY0real;
	END_IF;
	
	IF #tempYreal < #tempYminReal THEN
	    #SclScaleLinearRealToInt := 0;
	ELSIF #tempYreal > #tempYmaxReal THEN
	    #SclScaleLinearRealToInt := #yMax;
	ELSE
	    #SclScaleLinearRealToInt := REAL_TO_INT(#tempYreal);
	END_IF;
END_FUNCTION

FUNCTION "ERR_CompareGetErrorComponent" : Bool
{ S7_Optimized_Access := 'TRUE' }
VERSION : 0.1
   VAR_INPUT 
      Actual : "stt_ERR_ComponentGetError";
      Buffer : "stt_ERR_GetError";
   END_VAR

   VAR_TEMP 
      tempCounter : USInt;
   END_VAR


BEGIN
	#ERR_CompareGetErrorComponent := FALSE;
	//Get Counter value
	#tempCounter := #Buffer.Counter;
	//searching difference
	IF (#Buffer.Component[#tempCounter].BlockType <> #Actual.BlockType) THEN
	    #ERR_CompareGetErrorComponent := TRUE;
	ELSIF (#Buffer.Component[#tempCounter].BlockNumber <> #Actual.BlockNumber) THEN
	    #ERR_CompareGetErrorComponent := TRUE;
	ELSIF (#Buffer.Component[#tempCounter].MemoryArea <> #Actual.MemoryArea) THEN
	    #ERR_CompareGetErrorComponent := TRUE;
	ELSIF (#Buffer.Component[#tempCounter].NumberDB <> #Actual.NumberDB) THEN
	    #ERR_CompareGetErrorComponent := TRUE;
	END_IF;
	
END_FUNCTION

FUNCTION "ERR_GetSoftwareError" : Void
{ S7_Optimized_Access := 'TRUE' }
VERSION : 0.1
   VAR_INPUT 
      Error : Bool;
      Status : DWord;
   END_VAR

   VAR_IN_OUT 
      Buffer : "stt_ERR_SoftwareError";
   END_VAR


BEGIN
	IF (#Error = TRUE) THEN
	    IF ("ERR_CompareSoftwareError"(Actual := #Status, Buffer := #Buffer)) THEN
	        "ERR_OverflowBufferControl"(Counter := #Buffer.Counter,
	                                    Overflow := #Buffer.Overflow);
	        "ERR_SaveSoftwareErrorToBuffer"(DataToSave := #Status,
	                                        Buffer := #Buffer);
	    END_IF;
	END_IF;
	
	
END_FUNCTION

FUNCTION "ERR_OverflowBufferControl" : Void
{ S7_Optimized_Access := 'TRUE' }
VERSION : 0.1
   VAR_IN_OUT 
      "Counter" : USInt;
      Overflow : Bool;
   END_VAR


BEGIN
	#Counter := #Counter + 1;
	IF(#Counter > 4) THEN
	  #Counter := 0;
	  #Overflow := TRUE;
	END_IF;
	
END_FUNCTION

FUNCTION "ERR_SaveSoftwareErrorToBuffer" : Void
{ S7_Optimized_Access := 'TRUE' }
VERSION : 0.1
   VAR_INPUT 
      DataToSave : DWord;
   END_VAR

   VAR_IN_OUT 
      Buffer : "stt_ERR_SoftwareError";
   END_VAR

   VAR_TEMP 
      tempCounter : USInt;
   END_VAR


BEGIN
	//#tempCounter := #Buffer.Counter;
	#Buffer.Status[#Buffer.Counter] := #DataToSave;
END_FUNCTION

DATA_BLOCK "Alarm-Pompownia-Sucho-Max_DB"   // DB143
AUTHOR : rtecmer
VERSION : 0.1
// stored: AutoNumber true, DBAccessibleFromOPCUA true, InstanceOfName Alarm-Pompownia-Sucho-Max, InstanceOfType FB
"Alarm-Pompownia-Sucho-Max"
BEGIN
END_DATA_BLOCK

DATA_BLOCK "Alarm_min_magistrala_B5_DB"   // DB19
AUTHOR : rt69
VERSION : 0.1
// stored: AutoNumber true, DBAccessibleFromOPCUA true, InstanceOfName Alarm_min_magistrala_B5, InstanceOfType FB
"Alarm_min_magistrala_B5"
BEGIN
END_DATA_BLOCK

DATA_BLOCK "Strategia sterowaia Z11_DB_1"   // DB146
AUTHOR : rtecmer
VERSION : 0.1
// stored: AutoNumber true, DBAccessibleFromOPCUA true, InstanceOfName Strategia sterowaia Z11, InstanceOfType FB
"Strategia sterowaia Z11"
BEGIN
END_DATA_BLOCK

DATA_BLOCK "Strategia sterowaia Z12_DB"   // DB83
AUTHOR : rtecmer
VERSION : 0.1
// stored: AutoNumber true, DBAccessibleFromOPCUA true, InstanceOfName Strategia sterowaia Z12, InstanceOfType FB
"Strategia sterowaia Z12"
BEGIN
END_DATA_BLOCK

DATA_BLOCK "Control Current Overload_DB"   // DB72
AUTHOR : rtecmer
VERSION : 0.1
// stored: AutoNumber true, DBAccessibleFromOPCUA true, InstanceOfName Kontrola przeciążenia falownika, InstanceOfType FB
"Kontrola przeciążenia falownika"
BEGIN
END_DATA_BLOCK

DATA_BLOCK "ValueHz_in_Alarm_CurrentOver_DB"   // DB71
AUTHOR : rtecmer
VERSION : 0.1
// stored: AutoNumber true, DBAccessibleFromOPCUA true, InstanceOfName Kontrola Hz w trybie awayjnym od barMax, InstanceOfType FB
"Kontrola Hz w trybie awayjnym od barMax"
BEGIN
END_DATA_BLOCK

DATA_BLOCK "Byte Status Z11 Z12_DB"   // DB82
AUTHOR : rtecmer
VERSION : 0.1
// stored: AutoNumber true, DBAccessibleFromOPCUA true, InstanceOfName Byte status zasuw, InstanceOfType FB
"Byte status zasuw"
BEGIN
END_DATA_BLOCK

DATA_BLOCK "IEC_Counter_ControlAlarm_DB"   // DB73
{ S7_Optimized_Access := 'TRUE' }
// stored: AutoNumber false, DBAccessibleFromOPCUA true, InstanceOfName IEC_COUNTER, OfSystemLibElement IEC_COUNTER, OfSystemLibVersion 1.0
"IEC_COUNTER"
   // VAR RETAIN
   //    CU : Bool;
   //    CD : Bool;
   //    R : Bool;
   //    LD : Bool;
   //    QU : Bool;
   //    QD : Bool;
   //    PV : Int;
   //    CV : Int;
   // END_VAR
BEGIN
END_DATA_BLOCK

DATA_BLOCK "IEC_SetLimitFir1_0_DB"   // DB97
{ S7_Optimized_Access := 'TRUE' }
// stored: AutoNumber true, DBAccessibleFromOPCUA true, InstanceOfName IEC_TIMER, OfSystemLibElement IEC_TIMER, OfSystemLibVersion 1.0
"IEC_TIMER"
   // VAR
   //    PT : Time;
   //    ET { ExternalWritable := 'False'} : Time;
   //    IN : Bool;
   //    Q { ExternalWritable := 'False'} : Bool;
   // END_VAR
BEGIN
END_DATA_BLOCK

DATA_BLOCK "IEC_Timer1_Generator1Hz_DB"   // DB16
{ S7_Optimized_Access := 'TRUE' }
// stored: AutoNumber true, DBAccessibleFromOPCUA true, InstanceOfName IEC_TIMER, OfSystemLibElement IEC_TIMER, OfSystemLibVersion 1.0
"IEC_TIMER"
   // VAR
   //    PT : Time;
   //    ET { ExternalWritable := 'False'} : Time;
   //    IN : Bool;
   //    Q { ExternalWritable := 'False'} : Bool;
   // END_VAR
BEGIN
END_DATA_BLOCK

DATA_BLOCK "IEC_Timer2_Generator1Hz_DB"   // DB17
{ S7_Optimized_Access := 'TRUE' }
// stored: AutoNumber true, DBAccessibleFromOPCUA true, InstanceOfName IEC_TIMER, OfSystemLibElement IEC_TIMER, OfSystemLibVersion 1.0
"IEC_TIMER"
   // VAR
   //    PT : Time;
   //    ET { ExternalWritable := 'False'} : Time;
   //    IN : Bool;
   //    Q { ExternalWritable := 'False'} : Bool;
   // END_VAR
BEGIN
END_DATA_BLOCK

DATA_BLOCK "IEC_Timer_50Hz_DB"   // DB13
{ S7_Optimized_Access := 'TRUE' }
// stored: AutoNumber true, DBAccessibleFromOPCUA true, InstanceOfName IEC_TIMER, OfSystemLibElement IEC_TIMER, OfSystemLibVersion 1.0
"IEC_TIMER"
   // VAR
   //    PT : Time;
   //    ET { ExternalWritable := 'False'} : Time;
   //    IN : Bool;
   //    Q { ExternalWritable := 'False'} : Bool;
   // END_VAR
BEGIN
END_DATA_BLOCK

DATA_BLOCK "IEC_Timer_Ampere_Max_reset_DB"   // DB65
{ S7_Optimized_Access := 'TRUE' }
// stored: AutoNumber true, DBAccessibleFromOPCUA true, InstanceOfName IEC_TIMER, OfSystemLibElement IEC_TIMER, OfSystemLibVersion 1.0
"IEC_TIMER"
   // VAR
   //    PT : Time;
   //    ET { ExternalWritable := 'False'} : Time;
   //    IN : Bool;
   //    Q { ExternalWritable := 'False'} : Bool;
   // END_VAR
BEGIN
END_DATA_BLOCK

DATA_BLOCK "IEC_Timer_B7max_bar_DB"   // DB117
{ S7_Optimized_Access := 'TRUE' }
// stored: AutoNumber true, DBAccessibleFromOPCUA true, InstanceOfName IEC_TIMER, OfSystemLibElement IEC_TIMER, OfSystemLibVersion 1.0
"IEC_TIMER"
   // VAR
   //    PT : Time;
   //    ET { ExternalWritable := 'False'} : Time;
   //    IN : Bool;
   //    Q { ExternalWritable := 'False'} : Bool;
   // END_VAR
BEGIN
END_DATA_BLOCK

DATA_BLOCK "IEC_Timer_B7max_off_alarm_DB"   // DB142
{ S7_Optimized_Access := 'TRUE' }
// stored: AutoNumber true, DBAccessibleFromOPCUA true, InstanceOfName IEC_TIMER, OfSystemLibElement IEC_TIMER, OfSystemLibVersion 1.0
"IEC_TIMER"
   // VAR
   //    PT : Time;
   //    ET { ExternalWritable := 'False'} : Time;
   //    IN : Bool;
   //    Q { ExternalWritable := 'False'} : Bool;
   // END_VAR
BEGIN
END_DATA_BLOCK

DATA_BLOCK "IEC_Timer_Hist_SetHWork_P1_DB"   // DB43
{ S7_Optimized_Access := 'TRUE' }
// stored: AutoNumber true, DBAccessibleFromOPCUA true, InstanceOfName IEC_TIMER, OfSystemLibElement IEC_TIMER, OfSystemLibVersion 1.0
"IEC_TIMER"
   // VAR
   //    PT : Time;
   //    ET { ExternalWritable := 'False'} : Time;
   //    IN : Bool;
   //    Q { ExternalWritable := 'False'} : Bool;
   // END_VAR
BEGIN
END_DATA_BLOCK

DATA_BLOCK "IEC_Timer_Hist_SetHWork_P2_DB"   // DB44
{ S7_Optimized_Access := 'TRUE' }
// stored: AutoNumber true, DBAccessibleFromOPCUA true, InstanceOfName IEC_TIMER, OfSystemLibElement IEC_TIMER, OfSystemLibVersion 1.0
"IEC_TIMER"
   // VAR
   //    PT : Time;
   //    ET { ExternalWritable := 'False'} : Time;
   //    IN : Bool;
   //    Q { ExternalWritable := 'False'} : Bool;
   // END_VAR
BEGIN
END_DATA_BLOCK

DATA_BLOCK "IEC_Timer_Hist_SetHWork_P3_DB"   // DB45
{ S7_Optimized_Access := 'TRUE' }
// stored: AutoNumber true, DBAccessibleFromOPCUA true, InstanceOfName IEC_TIMER, OfSystemLibElement IEC_TIMER, OfSystemLibVersion 1.0
"IEC_TIMER"
   // VAR
   //    PT : Time;
   //    ET { ExternalWritable := 'False'} : Time;
   //    IN : Bool;
   //    Q { ExternalWritable := 'False'} : Bool;
   // END_VAR
BEGIN
END_DATA_BLOCK

DATA_BLOCK "IEC_Timer_Hist_SetHWork_P4_DB"   // DB28
{ S7_Optimized_Access := 'TRUE' }
// stored: AutoNumber true, DBAccessibleFromOPCUA true, InstanceOfName IEC_TIMER, OfSystemLibElement IEC_TIMER, OfSystemLibVersion 1.0
"IEC_TIMER"
   // VAR
   //    PT : Time;
   //    ET { ExternalWritable := 'False'} : Time;
   //    IN : Bool;
   //    Q { ExternalWritable := 'False'} : Bool;
   // END_VAR
BEGIN
END_DATA_BLOCK

DATA_BLOCK "IEC_Timer_HisterRresetNetwork50hz_DB"   // DB94
{ S7_Optimized_Access := 'TRUE' }
// stored: AutoNumber true, DBAccessibleFromOPCUA true, InstanceOfName IEC_TIMER, OfSystemLibElement IEC_TIMER, OfSystemLibVersion 1.0
"IEC_TIMER"
   // VAR
   //    PT : Time;
   //    ET { ExternalWritable := 'False'} : Time;
   //    IN : Bool;
   //    Q { ExternalWritable := 'False'} : Bool;
   // END_VAR
BEGIN
END_DATA_BLOCK

DATA_BLOCK "IEC_Timer_InputWarningH_DB"   // DB96
{ S7_Optimized_Access := 'TRUE' }
// stored: AutoNumber true, DBAccessibleFromOPCUA true, InstanceOfName IEC_TIMER, OfSystemLibElement IEC_TIMER, OfSystemLibVersion 1.0
"IEC_TIMER"
   // VAR
   //    PT : Time;
   //    ET { ExternalWritable := 'False'} : Time;
   //    IN : Bool;
   //    Q { ExternalWritable := 'False'} : Bool;
   // END_VAR
BEGIN
END_DATA_BLOCK

DATA_BLOCK "IEC_Timer_K1OFF_DB"   // DB11
{ S7_Optimized_Access := 'TRUE' }
// stored: AutoNumber true, DBAccessibleFromOPCUA true, InstanceOfName IEC_TIMER, OfSystemLibElement IEC_TIMER, OfSystemLibVersion 1.0
"IEC_TIMER"
   // VAR
   //    PT : Time;
   //    ET { ExternalWritable := 'False'} : Time;
   //    IN : Bool;
   //    Q { ExternalWritable := 'False'} : Bool;
   // END_VAR
BEGIN
END_DATA_BLOCK

DATA_BLOCK "IEC_Timer_K1ON_DB"   // DB12
{ S7_Optimized_Access := 'TRUE' }
// stored: AutoNumber true, DBAccessibleFromOPCUA true, InstanceOfName IEC_TIMER, OfSystemLibElement IEC_TIMER, OfSystemLibVersion 1.0
"IEC_TIMER"
   // VAR
   //    PT : Time;
   //    ET { ExternalWritable := 'False'} : Time;
   //    IN : Bool;
   //    Q { ExternalWritable := 'False'} : Bool;
   // END_VAR
BEGIN
END_DATA_BLOCK

DATA_BLOCK "IEC_Timer_K2OFF_DB"   // DB8
{ S7_Optimized_Access := 'TRUE' }
// stored: AutoNumber true, DBAccessibleFromOPCUA true, InstanceOfName IEC_TIMER, OfSystemLibElement IEC_TIMER, OfSystemLibVersion 1.0
"IEC_TIMER"
   // VAR
   //    PT : Time;
   //    ET { ExternalWritable := 'False'} : Time;
   //    IN : Bool;
   //    Q { ExternalWritable := 'False'} : Bool;
   // END_VAR
BEGIN
END_DATA_BLOCK

DATA_BLOCK "IEC_Timer_K2ON_DB"   // DB9
{ S7_Optimized_Access := 'TRUE' }
// stored: AutoNumber true, DBAccessibleFromOPCUA true, InstanceOfName IEC_TIMER, OfSystemLibElement IEC_TIMER, OfSystemLibVersion 1.0
"IEC_TIMER"
   // VAR
   //    PT : Time;
   //    ET { ExternalWritable := 'False'} : Time;
   //    IN : Bool;
   //    Q { ExternalWritable := 'False'} : Bool;
   // END_VAR
BEGIN
END_DATA_BLOCK

DATA_BLOCK "IEC_Timer_K3OFF_DB"   // DB26
{ S7_Optimized_Access := 'TRUE' }
// stored: AutoNumber true, DBAccessibleFromOPCUA true, InstanceOfName IEC_TIMER, OfSystemLibElement IEC_TIMER, OfSystemLibVersion 1.0
"IEC_TIMER"
   // VAR
   //    PT : Time;
   //    ET { ExternalWritable := 'False'} : Time;
   //    IN : Bool;
   //    Q { ExternalWritable := 'False'} : Bool;
   // END_VAR
BEGIN
END_DATA_BLOCK

DATA_BLOCK "IEC_Timer_K3ON_DB"   // DB25
{ S7_Optimized_Access := 'TRUE' }
// stored: AutoNumber true, DBAccessibleFromOPCUA true, InstanceOfName IEC_TIMER, OfSystemLibElement IEC_TIMER, OfSystemLibVersion 1.0
"IEC_TIMER"
   // VAR
   //    PT : Time;
   //    ET { ExternalWritable := 'False'} : Time;
   //    IN : Bool;
   //    Q { ExternalWritable := 'False'} : Bool;
   // END_VAR
BEGIN
END_DATA_BLOCK

DATA_BLOCK "IEC_Timer_OpenZ11_strategia_DB"   // DB130
{ S7_Optimized_Access := 'TRUE' }
// stored: AutoNumber true, DBAccessibleFromOPCUA true, InstanceOfName IEC_TIMER, OfSystemLibElement IEC_TIMER, OfSystemLibVersion 1.0
"IEC_TIMER"
   // VAR
   //    PT : Time;
   //    ET { ExternalWritable := 'False'} : Time;
   //    IN : Bool;
   //    Q { ExternalWritable := 'False'} : Bool;
   // END_VAR
BEGIN
END_DATA_BLOCK

DATA_BLOCK "IEC_Timer_OpenZ12_DB"   // DB135
{ S7_Optimized_Access := 'TRUE' }
// stored: AutoNumber true, DBAccessibleFromOPCUA true, InstanceOfName IEC_TIMER, OfSystemLibElement IEC_TIMER, OfSystemLibVersion 1.0
"IEC_TIMER"
   // VAR
   //    PT : Time;
   //    ET { ExternalWritable := 'False'} : Time;
   //    IN : Bool;
   //    Q { ExternalWritable := 'False'} : Bool;
   // END_VAR
BEGIN
END_DATA_BLOCK

DATA_BLOCK "IEC_Timer_P1_ready_DB"   // DB133
{ S7_Optimized_Access := 'TRUE' }
// stored: AutoNumber true, DBAccessibleFromOPCUA true, InstanceOfName IEC_TIMER, OfSystemLibElement IEC_TIMER, OfSystemLibVersion 1.0
"IEC_TIMER"
   // VAR
   //    PT : Time;
   //    ET { ExternalWritable := 'False'} : Time;
   //    IN : Bool;
   //    Q { ExternalWritable := 'False'} : Bool;
   // END_VAR
BEGIN
END_DATA_BLOCK

DATA_BLOCK "IEC_Timer_P2_ready_DB"   // DB144
{ S7_Optimized_Access := 'TRUE' }
// stored: AutoNumber true, DBAccessibleFromOPCUA true, InstanceOfName IEC_TIMER, OfSystemLibElement IEC_TIMER, OfSystemLibVersion 1.0
"IEC_TIMER"
   // VAR
   //    PT : Time;
   //    ET { ExternalWritable := 'False'} : Time;
   //    IN : Bool;
   //    Q { ExternalWritable := 'False'} : Bool;
   // END_VAR
BEGIN
END_DATA_BLOCK

DATA_BLOCK "IEC_Timer_P3_ready_DB"   // DB145
{ S7_Optimized_Access := 'TRUE' }
// stored: AutoNumber true, DBAccessibleFromOPCUA true, InstanceOfName IEC_TIMER, OfSystemLibElement IEC_TIMER, OfSystemLibVersion 1.0
"IEC_TIMER"
   // VAR
   //    PT : Time;
   //    ET { ExternalWritable := 'False'} : Time;
   //    IN : Bool;
   //    Q { ExternalWritable := 'False'} : Bool;
   // END_VAR
BEGIN
END_DATA_BLOCK

DATA_BLOCK "IEC_Timer_P4_ready_DB"   // DB147
{ S7_Optimized_Access := 'TRUE' }
// stored: AutoNumber true, DBAccessibleFromOPCUA true, InstanceOfName IEC_TIMER, OfSystemLibElement IEC_TIMER, OfSystemLibVersion 1.0
"IEC_TIMER"
   // VAR
   //    PT : Time;
   //    ET { ExternalWritable := 'False'} : Time;
   //    IN : Bool;
   //    Q { ExternalWritable := 'False'} : Bool;
   // END_VAR
BEGIN
END_DATA_BLOCK

DATA_BLOCK "IEC_Timer_PressO2_Max_DB"   // DB63
{ S7_Optimized_Access := 'TRUE' }
// stored: AutoNumber true, DBAccessibleFromOPCUA true, InstanceOfName IEC_TIMER, OfSystemLibElement IEC_TIMER, OfSystemLibVersion 1.0
"IEC_TIMER"
   // VAR
   //    PT : Time;
   //    ET { ExternalWritable := 'False'} : Time;
   //    IN : Bool;
   //    Q { ExternalWritable := 'False'} : Bool;
   // END_VAR
BEGIN
END_DATA_BLOCK

DATA_BLOCK "IEC_Timer_ResK1errorRun_DB"   // DB101
{ S7_Optimized_Access := 'TRUE' }
// stored: AutoNumber true, DBAccessibleFromOPCUA true, InstanceOfName IEC_TIMER, OfSystemLibElement IEC_TIMER, OfSystemLibVersion 1.0
"IEC_TIMER"
   // VAR
   //    PT : Time;
   //    ET { ExternalWritable := 'False'} : Time;
   //    IN : Bool;
   //    Q { ExternalWritable := 'False'} : Bool;
   // END_VAR
BEGIN
END_DATA_BLOCK

DATA_BLOCK "IEC_Timer_ResetPID_stst0_DB"   // DB20
{ S7_Optimized_Access := 'TRUE' }
// stored: AutoNumber true, DBAccessibleFromOPCUA true, InstanceOfName IEC_TIMER, OfSystemLibElement IEC_TIMER, OfSystemLibVersion 1.0
"IEC_TIMER"
   // VAR
   //    PT : Time;
   //    ET { ExternalWritable := 'False'} : Time;
   //    IN : Bool;
   //    Q { ExternalWritable := 'False'} : Bool;
   // END_VAR
BEGIN
END_DATA_BLOCK

DATA_BLOCK "IEC_Timer_Reset_Is_Up_Hz_DB"   // DB50
{ S7_Optimized_Access := 'TRUE' }
// stored: AutoNumber true, DBAccessibleFromOPCUA true, InstanceOfName IEC_TIMER, OfSystemLibElement IEC_TIMER, OfSystemLibVersion 1.0
"IEC_TIMER"
   // VAR
   //    PT : Time;
   //    ET { ExternalWritable := 'False'} : Time;
   //    IN : Bool;
   //    Q { ExternalWritable := 'False'} : Bool;
   // END_VAR
BEGIN
END_DATA_BLOCK

DATA_BLOCK "IEC_Timer_Reset_Set_Motor2_DB"   // DB75
{ S7_Optimized_Access := 'TRUE' }
// stored: AutoNumber true, DBAccessibleFromOPCUA true, InstanceOfName IEC_TIMER, OfSystemLibElement IEC_TIMER, OfSystemLibVersion 1.0
"IEC_TIMER"
   // VAR
   //    PT : Time;
   //    ET { ExternalWritable := 'False'} : Time;
   //    IN : Bool;
   //    Q { ExternalWritable := 'False'} : Bool;
   // END_VAR
BEGIN
END_DATA_BLOCK

DATA_BLOCK "IEC_Timer_Reset_Set_Motor3_DB"   // DB93
{ S7_Optimized_Access := 'TRUE' }
// stored: AutoNumber true, DBAccessibleFromOPCUA true, InstanceOfName IEC_TIMER, OfSystemLibElement IEC_TIMER, OfSystemLibVersion 1.0
"IEC_TIMER"
   // VAR
   //    PT : Time;
   //    ET { ExternalWritable := 'False'} : Time;
   //    IN : Bool;
   //    Q { ExternalWritable := 'False'} : Bool;
   // END_VAR
BEGIN
END_DATA_BLOCK

DATA_BLOCK "IEC_Timer_Reset_Set_Motor4_DB"   // DB84
{ S7_Optimized_Access := 'TRUE' }
// stored: AutoNumber true, DBAccessibleFromOPCUA true, InstanceOfName IEC_TIMER, OfSystemLibElement IEC_TIMER, OfSystemLibVersion 1.0
"IEC_TIMER"
   // VAR
   //    PT : Time;
   //    ET { ExternalWritable := 'False'} : Time;
   //    IN : Bool;
   //    Q { ExternalWritable := 'False'} : Bool;
   // END_VAR
BEGIN
END_DATA_BLOCK

DATA_BLOCK "IEC_Timer_Reset_delay_DB"   // DB67
{ S7_Optimized_Access := 'TRUE' }
// stored: AutoNumber true, DBAccessibleFromOPCUA true, InstanceOfName IEC_TIMER, OfSystemLibElement IEC_TIMER, OfSystemLibVersion 1.0
"IEC_TIMER"
   // VAR
   //    PT : Time;
   //    ET { ExternalWritable := 'False'} : Time;
   //    IN : Bool;
   //    Q { ExternalWritable := 'False'} : Bool;
   // END_VAR
BEGIN
END_DATA_BLOCK

DATA_BLOCK "IEC_Timer_SUPV_SM_DB"   // DB95
{ S7_Optimized_Access := 'TRUE' }
// stored: AutoNumber true, DBAccessibleFromOPCUA true, InstanceOfName IEC_TIMER, OfSystemLibElement IEC_TIMER, OfSystemLibVersion 1.0
"IEC_TIMER"
   // VAR
   //    PT : Time;
   //    ET { ExternalWritable := 'False'} : Time;
   //    IN : Bool;
   //    Q { ExternalWritable := 'False'} : Bool;
   // END_VAR
BEGIN
END_DATA_BLOCK

DATA_BLOCK "IEC_Timer_Set_50Hz_DB"   // DB66
{ S7_Optimized_Access := 'TRUE' }
// stored: AutoNumber true, DBAccessibleFromOPCUA true, InstanceOfName IEC_TIMER, OfSystemLibElement IEC_TIMER, OfSystemLibVersion 1.0
"IEC_TIMER"
   // VAR
   //    PT : Time;
   //    ET { ExternalWritable := 'False'} : Time;
   //    IN : Bool;
   //    Q { ExternalWritable := 'False'} : Bool;
   // END_VAR
BEGIN
END_DATA_BLOCK

DATA_BLOCK "IEC_Timer_Set_Current_Overload_InverterKDN_DB"   // DB68
{ S7_Optimized_Access := 'TRUE' }
// stored: AutoNumber true, DBAccessibleFromOPCUA true, InstanceOfName IEC_TIMER, OfSystemLibElement IEC_TIMER, OfSystemLibVersion 1.0
"IEC_TIMER"
   // VAR
   //    PT : Time;
   //    ET { ExternalWritable := 'False'} : Time;
   //    IN : Bool;
   //    Q { ExternalWritable := 'False'} : Bool;
   // END_VAR
BEGIN
END_DATA_BLOCK

DATA_BLOCK "IEC_Timer_Start-InverterP2_DB"   // DB40
{ S7_Optimized_Access := 'TRUE' }
// stored: AutoNumber true, DBAccessibleFromOPCUA true, InstanceOfName IEC_TIMER, OfSystemLibElement IEC_TIMER, OfSystemLibVersion 1.0
"IEC_TIMER"
   // VAR
   //    PT : Time;
   //    ET { ExternalWritable := 'False'} : Time;
   //    IN : Bool;
   //    Q { ExternalWritable := 'False'} : Bool;
   // END_VAR
BEGIN
END_DATA_BLOCK

DATA_BLOCK "IEC_Timer_Start-InverterP3_DB"   // DB41
{ S7_Optimized_Access := 'TRUE' }
// stored: AutoNumber true, DBAccessibleFromOPCUA true, InstanceOfName IEC_TIMER, OfSystemLibElement IEC_TIMER, OfSystemLibVersion 1.0
"IEC_TIMER"
   // VAR
   //    PT : Time;
   //    ET { ExternalWritable := 'False'} : Time;
   //    IN : Bool;
   //    Q { ExternalWritable := 'False'} : Bool;
   // END_VAR
BEGIN
END_DATA_BLOCK

DATA_BLOCK "IEC_Timer_Start-InverterP4_DB"   // DB27
{ S7_Optimized_Access := 'TRUE' }
// stored: AutoNumber true, DBAccessibleFromOPCUA true, InstanceOfName IEC_TIMER, OfSystemLibElement IEC_TIMER, OfSystemLibVersion 1.0
"IEC_TIMER"
   // VAR
   //    PT : Time;
   //    ET { ExternalWritable := 'False'} : Time;
   //    IN : Bool;
   //    Q { ExternalWritable := 'False'} : Bool;
   // END_VAR
BEGIN
END_DATA_BLOCK

DATA_BLOCK "IEC_Timer_Start_InverterP1_DB"   // DB39
{ S7_Optimized_Access := 'TRUE' }
// stored: AutoNumber true, DBAccessibleFromOPCUA true, InstanceOfName IEC_TIMER, OfSystemLibElement IEC_TIMER, OfSystemLibVersion 1.0
"IEC_TIMER"
   // VAR
   //    PT : Time;
   //    ET { ExternalWritable := 'False'} : Time;
   //    IN : Bool;
   //    Q { ExternalWritable := 'False'} : Bool;
   // END_VAR
BEGIN
END_DATA_BLOCK

DATA_BLOCK "IEC_Timer_TCP_conected_DB"   // DB113
{ S7_Optimized_Access := 'TRUE' }
// stored: AutoNumber true, DBAccessibleFromOPCUA true, InstanceOfName IEC_TIMER, OfSystemLibElement IEC_TIMER, OfSystemLibVersion 1.0
"IEC_TIMER"
   // VAR
   //    PT : Time;
   //    ET { ExternalWritable := 'False'} : Time;
   //    IN : Bool;
   //    Q { ExternalWritable := 'False'} : Bool;
   // END_VAR
BEGIN
END_DATA_BLOCK

DATA_BLOCK "IEC_Timer_WatchDogWicc-PLC_DB"   // DB22
{ S7_Optimized_Access := 'TRUE' }
// stored: AutoNumber true, DBAccessibleFromOPCUA true, InstanceOfName IEC_TIMER, OfSystemLibElement IEC_TIMER, OfSystemLibVersion 1.0
"IEC_TIMER"
   // VAR
   //    PT : Time;
   //    ET { ExternalWritable := 'False'} : Time;
   //    IN : Bool;
   //    Q { ExternalWritable := 'False'} : Bool;
   // END_VAR
BEGIN
END_DATA_BLOCK

DATA_BLOCK "IEC_Timer_WatchDogWinCC_cd_DB"   // DB23
{ S7_Optimized_Access := 'TRUE' }
// stored: AutoNumber true, DBAccessibleFromOPCUA true, InstanceOfName IEC_TIMER, OfSystemLibElement IEC_TIMER, OfSystemLibVersion 1.0
"IEC_TIMER"
   // VAR
   //    PT : Time;
   //    ET { ExternalWritable := 'False'} : Time;
   //    IN : Bool;
   //    Q { ExternalWritable := 'False'} : Bool;
   // END_VAR
BEGIN
END_DATA_BLOCK

DATA_BLOCK "IEC_Timer_WorningH_O2__DB"   // DB99
{ S7_Optimized_Access := 'TRUE' }
// stored: AutoNumber true, DBAccessibleFromOPCUA true, InstanceOfName IEC_TIMER, OfSystemLibElement IEC_TIMER, OfSystemLibVersion 1.0
"IEC_TIMER"
   // VAR
   //    PT : Time;
   //    ET { ExternalWritable := 'False'} : Time;
   //    IN : Bool;
   //    Q { ExternalWritable := 'False'} : Bool;
   // END_VAR
BEGIN
END_DATA_BLOCK

DATA_BLOCK "IEC_Timer_ZamykanieZ12_DB"   // DB136
{ S7_Optimized_Access := 'TRUE' }
// stored: AutoNumber true, DBAccessibleFromOPCUA true, InstanceOfName IEC_TIMER, OfSystemLibElement IEC_TIMER, OfSystemLibVersion 1.0
"IEC_TIMER"
   // VAR
   //    PT : Time;
   //    ET { ExternalWritable := 'False'} : Time;
   //    IN : Bool;
   //    Q { ExternalWritable := 'False'} : Bool;
   // END_VAR
BEGIN
END_DATA_BLOCK

DATA_BLOCK "IEC_Timer_Zmykanie Z11_DB"   // DB134
{ S7_Optimized_Access := 'TRUE' }
// stored: AutoNumber true, DBAccessibleFromOPCUA true, InstanceOfName IEC_TIMER, OfSystemLibElement IEC_TIMER, OfSystemLibVersion 1.0
"IEC_TIMER"
   // VAR
   //    PT : Time;
   //    ET { ExternalWritable := 'False'} : Time;
   //    IN : Bool;
   //    Q { ExternalWritable := 'False'} : Bool;
   // END_VAR
BEGIN
END_DATA_BLOCK

DATA_BLOCK "IEC_Timer_alarm_reset_DB"   // DB98
{ S7_Optimized_Access := 'TRUE' }
// stored: AutoNumber true, DBAccessibleFromOPCUA true, InstanceOfName IEC_TIMER, OfSystemLibElement IEC_TIMER, OfSystemLibVersion 1.0
"IEC_TIMER"
   // VAR
   //    PT : Time;
   //    ET { ExternalWritable := 'False'} : Time;
   //    IN : Bool;
   //    Q { ExternalWritable := 'False'} : Bool;
   // END_VAR
BEGIN
END_DATA_BLOCK

DATA_BLOCK "IEC_Timer_errorRTU_histereza_DB"   // DB129
{ S7_Optimized_Access := 'TRUE' }
// stored: AutoNumber true, DBAccessibleFromOPCUA true, InstanceOfName IEC_TIMER, OfSystemLibElement IEC_TIMER, OfSystemLibVersion 1.0
"IEC_TIMER"
   // VAR
   //    PT : Time;
   //    ET { ExternalWritable := 'False'} : Time;
   //    IN : Bool;
   //    Q { ExternalWritable := 'False'} : Bool;
   // END_VAR
BEGIN
END_DATA_BLOCK

DATA_BLOCK "IEC_Timer_resDodtkowa_DB"   // DB111
{ S7_Optimized_Access := 'TRUE' }
// stored: AutoNumber true, DBAccessibleFromOPCUA true, InstanceOfName IEC_TIMER, OfSystemLibElement IEC_TIMER, OfSystemLibVersion 1.0
"IEC_TIMER"
   // VAR
   //    PT : Time;
   //    ET { ExternalWritable := 'False'} : Time;
   //    IN : Bool;
   //    Q { ExternalWritable := 'False'} : Bool;
   // END_VAR
BEGIN
END_DATA_BLOCK

DATA_BLOCK "IEC_Timer_reset_conected_server TCP_DB"   // DB141
{ S7_Optimized_Access := 'TRUE' }
// stored: AutoNumber true, DBAccessibleFromOPCUA true, InstanceOfName IEC_TIMER, OfSystemLibElement IEC_TIMER, OfSystemLibVersion 1.0
"IEC_TIMER"
   // VAR
   //    PT : Time;
   //    ET { ExternalWritable := 'False'} : Time;
   //    IN : Bool;
   //    Q { ExternalWritable := 'False'} : Bool;
   // END_VAR
BEGIN
END_DATA_BLOCK

DATA_BLOCK "IEC_Timer_tmp_up_reset_DB"   // DB140
{ S7_Optimized_Access := 'TRUE' }
// stored: AutoNumber true, DBAccessibleFromOPCUA true, InstanceOfName IEC_TIMER, OfSystemLibElement IEC_TIMER, OfSystemLibVersion 1.0
"IEC_TIMER"
   // VAR
   //    PT : Time;
   //    ET { ExternalWritable := 'False'} : Time;
   //    IN : Bool;
   //    Q { ExternalWritable := 'False'} : Bool;
   // END_VAR
BEGIN
END_DATA_BLOCK

DATA_BLOCK "MB_COMM_LOAD_DB"   // DB34
// stored: AutoNumber true, DBAccessibleFromOPCUA true, InstanceOfName MB_COMM_LOAD, OfSystemLibElement MB_COMM_LOAD, OfSystemLibVersion 2.1
"MB_COMM_LOAD"
   // VAR_INPUT
   //    REQ : Bool;
   //    PORT : PORT;
   //    BAUD : UDInt;
   //    PARITY : UInt;
   //    FLOW_CTRL : UInt;
   //    RTS_ON_DLY : UInt;
   //    RTS_OFF_DLY : UInt;
   //    RESP_TO : UInt;
   // END_VAR
   // VAR_OUTPUT
   //    DONE : Bool;
   //    ERROR : Bool;
   //    STATUS : Word;
   // END_VAR
   // VAR_IN_OUT
   //    MB_DB : MB_BASE;
   // END_VAR
   // VAR
   //    ICHAR_GAP : UInt;
   //    RETRIES : UInt;
   //    WRREC_STATUS : Word;
   //    RDREC_STATUS : Word;
   //    SFC_STATUS : Word;
   //    Port_CFG_SFB : Array[0..25] of Byte;
   //    Send_CFG_SFB : Array[0..16] of Byte;
   //    Rcv_CFG_SFB : Array[0..60] of Byte;
   //    STOP_BITS : USInt := 2;
   // END_VAR
BEGIN
END_DATA_BLOCK

DATA_BLOCK "MB_COMM_LOAD_DB_Slave1"   // DB127
// stored: AutoNumber true, DBAccessibleFromOPCUA true, InstanceOfName MB_COMM_LOAD, OfSystemLibElement MB_COMM_LOAD, OfSystemLibVersion 2.1
"MB_COMM_LOAD"
   // VAR_INPUT
   //    REQ : Bool;
   //    PORT : PORT;
   //    BAUD : UDInt;
   //    PARITY : UInt;
   //    FLOW_CTRL : UInt;
   //    RTS_ON_DLY : UInt;
   //    RTS_OFF_DLY : UInt;
   //    RESP_TO : UInt;
   // END_VAR
   // VAR_OUTPUT
   //    DONE : Bool;
   //    ERROR : Bool;
   //    STATUS : Word;
   // END_VAR
   // VAR_IN_OUT
   //    MB_DB : MB_BASE;
   // END_VAR
   // VAR
   //    ICHAR_GAP : UInt;
   //    RETRIES : UInt;
   //    WRREC_STATUS : Word;
   //    RDREC_STATUS : Word;
   //    SFC_STATUS : Word;
   //    Port_CFG_SFB : Array[0..25] of Byte;
   //    Send_CFG_SFB : Array[0..16] of Byte;
   //    Rcv_CFG_SFB : Array[0..60] of Byte;
   //    STOP_BITS : USInt;
   // END_VAR
BEGIN
END_DATA_BLOCK

DATA_BLOCK "MB_MASTER_DB"   // DB36
// stored: AutoNumber true, DBAccessibleFromOPCUA true, InstanceOfName MB_MASTER, OfSystemLibElement MB_MASTER, OfSystemLibVersion 2.2
"MB_MASTER"
   // // inherited from MB_BASE
   // VAR
   //    S_PORT : UInt;
   //    S_RESP_TO : UInt;
   //    S_ICHAR_GAP : UInt;
   //    S_RETRIES : UInt;
   // END_VAR
   // VAR_INPUT
   //    REQ : Bool;
   //    MB_ADDR : UInt;
   //    MODE : USInt;
   //    DATA_ADDR : UDInt;
   //    DATA_LEN : UInt;
   // END_VAR
   // VAR_OUTPUT
   //    DONE : Bool;
   //    BUSY : Bool;
   //    ERROR : Bool;
   //    STATUS : Word;
   // END_VAR
   // VAR_IN_OUT
   //    DATA_PTR : Variant;
   // END_VAR
   // VAR
   //    SEND_PTP_SFB : Array[0..11] of Byte;
   //    RCV_PTP_SFB : Array[0..11] of Byte;
   //    RCV_RST_SFB : Array[0..9] of Byte;
   //    PF_FREQUENCY : Real;
   //    BLOCKED_PROC_TIMEOUT : Real;
   //    CURRENT_TIME_VALUE : UDInt;
   //    SAVED_TIME_VALUE : UDInt;
   //    SAVED_SLAVE_ADDR : Word;
   //    SAVED_MODE : Word;
   //    SAVED_DATA_ADDR : DWord;
   //    SAVED_DATA_LEN : UInt;
   //    MB_STATE : UInt;
   //    COMM_SENT_COUNT : UInt;
   //    BYTE_COUNT : USInt;
   //    INIT_OK : Bool;
   //    ACTIVE : Bool;
   //    BROADCAST_FLAG : Bool;
   //    EXTENDED_ADDRESSING : Bool;
   //    SAVED_START_ADDR : UInt;
   //    TXBuf_Function_Offset : UDInt;
   //    TXBuf_Address_Offset : UDInt;
   //    TXBuf_Quantity_Offset : UDInt;
   // END_VAR
BEGIN
END_DATA_BLOCK

DATA_BLOCK "MB_SERVER_DB"   // DB85
// stored: AutoNumber true, DBAccessibleFromOPCUA true, InstanceOfName MB_SERVER, OfSystemLibElement MB_SERVER, OfSystemLibVersion 3.1
"MB_SERVER"
   // VAR_INPUT
   //    DISCONNECT : Bool;
   //    CONNECT_ID : UInt;
   //    IP_PORT : UInt;
   // END_VAR
   // VAR_OUTPUT
   //    NDR : Bool;
   //    DR : Bool;
   //    ERROR : Bool;
   //    STATUS : Word;
   // END_VAR
   // VAR_IN_OUT
   //    MB_HOLD_REG : Variant;
   // END_VAR
   // VAR
   //    TCON_SFB { S7_SetPoint := 'True'} : TCON;
   //    TDISCON_SFB { S7_SetPoint := 'True'} : TDISCON;
   //    TSEND_SFB { S7_SetPoint := 'True'} : TSEND;
   //    TRCV_SFB { S7_SetPoint := 'True'} : TRCV;
   //    TCON_Param { S7_SetPoint := 'True'} : TCON_Param;
   //    MB_State : UInt;
   //    Request_Count : UInt;
   //    Server_Message_Count : UInt;
   //    Xmt_Rcv_Count : UInt;
   //    Exception_Count : UInt;
   //    Success_Count : UInt;
   //    SL_Status_Hold : UInt;
   //    HR_Start_Offset : UInt;
   //    Init_OK : Bool;
   //    SL_Error_State : Bool;
   //    Connected : Bool;
   //    XMT_Set_NDR : Bool;
   //    XMT_Set_DR : Bool;
   // END_VAR
BEGIN
END_DATA_BLOCK

DATA_BLOCK "MB_SERVER_DB_100"   // DB115
// stored: AutoNumber true, DBAccessibleFromOPCUA true, InstanceOfName MB_SERVER, OfSystemLibElement MB_SERVER, OfSystemLibVersion 3.1
"MB_SERVER"
   // VAR_INPUT
   //    DISCONNECT : Bool;
   //    CONNECT_ID : UInt;
   //    IP_PORT : UInt;
   // END_VAR
   // VAR_OUTPUT
   //    NDR : Bool;
   //    DR : Bool;
   //    ERROR : Bool;
   //    STATUS : Word;
   // END_VAR
   // VAR_IN_OUT
   //    MB_HOLD_REG : Variant;
   // END_VAR
   // VAR
   //    TCON_SFB { S7_SetPoint := 'True'} : TCON;
   //    TDISCON_SFB { S7_SetPoint := 'True'} : TDISCON;
   //    TSEND_SFB { S7_SetPoint := 'True'} : TSEND;
   //    TRCV_SFB { S7_SetPoint := 'True'} : TRCV;
   //    TCON_Param { S7_SetPoint := 'True'} : TCON_Param;
   //    MB_State : UInt;
   //    Request_Count : UInt;
   //    Server_Message_Count : UInt;
   //    Xmt_Rcv_Count : UInt;
   //    Exception_Count : UInt;
   //    Success_Count : UInt;
   //    SL_Status_Hold : UInt;
   //    HR_Start_Offset : UInt;
   //    Init_OK : Bool;
   //    SL_Error_State : Bool;
   //    Connected : Bool;
   //    XMT_Set_NDR : Bool;
   //    XMT_Set_DR : Bool;
   // END_VAR
BEGIN
END_DATA_BLOCK

DATA_BLOCK "MB_SERVER_DB_Czasy"   // DB48
// stored: AutoNumber true, DBAccessibleFromOPCUA true, InstanceOfName MB_SERVER, OfSystemLibElement MB_SERVER, OfSystemLibVersion 3.1
"MB_SERVER"
   // VAR_INPUT
   //    DISCONNECT : Bool;
   //    CONNECT_ID : UInt;
   //    IP_PORT : UInt;
   // END_VAR
   // VAR_OUTPUT
   //    NDR : Bool;
   //    DR : Bool;
   //    ERROR : Bool;
   //    STATUS : Word;
   // END_VAR
   // VAR_IN_OUT
   //    MB_HOLD_REG : Variant;
   // END_VAR
   // VAR
   //    TCON_SFB { S7_SetPoint := 'True'} : TCON;
   //    TDISCON_SFB { S7_SetPoint := 'True'} : TDISCON;
   //    TSEND_SFB { S7_SetPoint := 'True'} : TSEND;
   //    TRCV_SFB { S7_SetPoint := 'True'} : TRCV;
   //    TCON_Param { S7_SetPoint := 'True'} : TCON_Param;
   //    MB_State : UInt;
   //    Request_Count : UInt;
   //    Server_Message_Count : UInt;
   //    Xmt_Rcv_Count : UInt;
   //    Exception_Count : UInt;
   //    Success_Count : UInt;
   //    SL_Status_Hold : UInt;
   //    HR_Start_Offset : UInt;
   //    Init_OK : Bool;
   //    SL_Error_State : Bool;
   //    Connected : Bool;
   //    XMT_Set_NDR : Bool;
   //    XMT_Set_DR : Bool;
   // END_VAR
BEGIN
END_DATA_BLOCK

DATA_BLOCK "MB_SERVER_DB_parametry"   // DB88
// stored: AutoNumber true, DBAccessibleFromOPCUA true, InstanceOfName MB_SERVER, OfSystemLibElement MB_SERVER, OfSystemLibVersion 3.1
"MB_SERVER"
   // VAR_INPUT
   //    DISCONNECT : Bool;
   //    CONNECT_ID : UInt;
   //    IP_PORT : UInt;
   // END_VAR
   // VAR_OUTPUT
   //    NDR : Bool;
   //    DR : Bool;
   //    ERROR : Bool;
   //    STATUS : Word;
   // END_VAR
   // VAR_IN_OUT
   //    MB_HOLD_REG : Variant;
   // END_VAR
   // VAR
   //    TCON_SFB { S7_SetPoint := 'True'} : TCON;
   //    TDISCON_SFB { S7_SetPoint := 'True'} : TDISCON;
   //    TSEND_SFB { S7_SetPoint := 'True'} : TSEND;
   //    TRCV_SFB { S7_SetPoint := 'True'} : TRCV;
   //    TCON_Param { S7_SetPoint := 'True'} : TCON_Param;
   //    MB_State : UInt;
   //    Request_Count : UInt;
   //    Server_Message_Count : UInt;
   //    Xmt_Rcv_Count : UInt;
   //    Exception_Count : UInt;
   //    Success_Count : UInt;
   //    SL_Status_Hold : UInt;
   //    HR_Start_Offset : UInt;
   //    Init_OK : Bool;
   //    SL_Error_State : Bool;
   //    Connected : Bool;
   //    XMT_Set_NDR : Bool;
   //    XMT_Set_DR : Bool;
   // END_VAR
BEGIN
END_DATA_BLOCK

DATA_BLOCK "MB_SLAVE_RTU_DB"   // DB58
// stored: AutoNumber true, DBAccessibleFromOPCUA true, InstanceOfName MB_SLAVE, OfSystemLibElement MB_SLAVE, OfSystemLibVersion 2.1
"MB_SLAVE"
   // // inherited from MB_BASE
   // VAR
   //    S_PORT : UInt;
   //    S_RESP_TO : UInt;
   //    S_ICHAR_GAP : UInt;
   //    S_RETRIES : UInt;
   // END_VAR
   // VAR_INPUT
   //    MB_ADDR : UInt;
   // END_VAR
   // VAR_OUTPUT
   //    NDR : Bool;
   //    DR : Bool;
   //    ERROR : Bool;
   //    STATUS : Word;
   // END_VAR
   // VAR_IN_OUT
   //    MB_HOLD_REG : Variant;
   // END_VAR
   // VAR
   //    SEND_PTP_SFB : Array[0..11] of Byte;
   //    RCV_PTP_SFB : Array[0..11] of Byte;
   //    MB_State : Word;
   //    Request_Count : Word;
   //    Slave_Message_Count : Word;
   //    Bad_CRC_Count : Word;
   //    Broadcast_Count : Word;
   //    Exception_Count : Word;
   //    Success_Count : Word;
   //    SL_Status_Hold : Word;
   //    HR_Start_Offset : Word;
   //    Init_OK : Bool;
   //    Broadcast_Flag : Bool;
   //    SL_Error_State : Bool;
   //    Extended_Addressing : Bool;
   //    XMT_Set_NDR : Bool;
   //    XMT_Set_DR : Bool;
   // END_VAR
BEGIN
END_DATA_BLOCK

DATA_BLOCK "Modbus_TCP_DB"   // DB87
AUTHOR : rtecmer
VERSION : 0.1
// stored: AutoNumber true, DBAccessibleFromOPCUA true, InstanceOfName Modbus_TCP, InstanceOfType FB
"Modbus_TCP"
BEGIN
END_DATA_BLOCK

DATA_BLOCK "R_TRIG_DB_AUT_M1"   // DB118
// stored: AutoNumber true, DBAccessibleFromOPCUA true, InstanceOfName R_TRIG, OfSystemLibElement R_TRIG, OfSystemLibVersion 1.0
"R_TRIG"
   // VAR_INPUT
   //    CLK : Bool;
   // END_VAR
   // VAR_OUTPUT
   //    Q : Bool;
   // END_VAR
   // VAR
   //    Stat_Bit : Bool;
   // END_VAR
BEGIN
END_DATA_BLOCK

DATA_BLOCK "R_TRIG_DB_AUT_M2"   // DB120
// stored: AutoNumber true, DBAccessibleFromOPCUA true, InstanceOfName R_TRIG, OfSystemLibElement R_TRIG, OfSystemLibVersion 1.0
"R_TRIG"
   // VAR_INPUT
   //    CLK : Bool;
   // END_VAR
   // VAR_OUTPUT
   //    Q : Bool;
   // END_VAR
   // VAR
   //    Stat_Bit : Bool;
   // END_VAR
BEGIN
END_DATA_BLOCK

DATA_BLOCK "R_TRIG_DB_AUT_M3"   // DB121
// stored: AutoNumber true, DBAccessibleFromOPCUA true, InstanceOfName R_TRIG, OfSystemLibElement R_TRIG, OfSystemLibVersion 1.0
"R_TRIG"
   // VAR_INPUT
   //    CLK : Bool;
   // END_VAR
   // VAR_OUTPUT
   //    Q : Bool;
   // END_VAR
   // VAR
   //    Stat_Bit : Bool;
   // END_VAR
BEGIN
END_DATA_BLOCK

DATA_BLOCK "R_TRIG_DB_AUT_M4"   // DB122
// stored: AutoNumber true, DBAccessibleFromOPCUA true, InstanceOfName R_TRIG, OfSystemLibElement R_TRIG, OfSystemLibVersion 1.0
"R_TRIG"
   // VAR_INPUT
   //    CLK : Bool;
   // END_VAR
   // VAR_OUTPUT
   //    Q : Bool;
   // END_VAR
   // VAR
   //    Stat_Bit : Bool;
   // END_VAR
BEGIN
END_DATA_BLOCK

DATA_BLOCK "R_TRIG_DB_AUT_Z11"   // DB123
// stored: AutoNumber true, DBAccessibleFromOPCUA true, InstanceOfName R_TRIG, OfSystemLibElement R_TRIG, OfSystemLibVersion 1.0
"R_TRIG"
   // VAR_INPUT
   //    CLK : Bool;
   // END_VAR
   // VAR_OUTPUT
   //    Q : Bool;
   // END_VAR
   // VAR
   //    Stat_Bit : Bool;
   // END_VAR
BEGIN
END_DATA_BLOCK

DATA_BLOCK "R_TRIG_DB_AUT_Z12"   // DB124
// stored: AutoNumber true, DBAccessibleFromOPCUA true, InstanceOfName R_TRIG, OfSystemLibElement R_TRIG, OfSystemLibVersion 1.0
"R_TRIG"
   // VAR_INPUT
   //    CLK : Bool;
   // END_VAR
   // VAR_OUTPUT
   //    Q : Bool;
   // END_VAR
   // VAR
   //    Stat_Bit : Bool;
   // END_VAR
BEGIN
END_DATA_BLOCK

DATA_BLOCK "R_TRIG_DB_CLK"   // DB126
// stored: AutoNumber true, DBAccessibleFromOPCUA true, InstanceOfName R_TRIG, OfSystemLibElement R_TRIG, OfSystemLibVersion 1.0
"R_TRIG"
   // VAR_INPUT
   //    CLK : Bool;
   // END_VAR
   // VAR_OUTPUT
   //    Q : Bool;
   // END_VAR
   // VAR
   //    Stat_Bit : Bool;
   // END_VAR
BEGIN
END_DATA_BLOCK

DATA_BLOCK "R_TRIG_DB_przechwycenie_strategii"   // DB138
// stored: AutoNumber true, DBAccessibleFromOPCUA true, InstanceOfName R_TRIG, OfSystemLibElement R_TRIG, OfSystemLibVersion 1.0
"R_TRIG"
   // VAR_INPUT
   //    CLK : Bool;
   // END_VAR
   // VAR_OUTPUT
   //    Q : Bool;
   // END_VAR
   // VAR
   //    Stat_Bit : Bool;
   // END_VAR
BEGIN
END_DATA_BLOCK

DATA_BLOCK "Strategia sterowania POMPOWNIA_DB"   // DB139
AUTHOR : rtecmer
VERSION : 0.1
// stored: AutoNumber true, DBAccessibleFromOPCUA true, InstanceOfName Strategia sterowania Pompownia, InstanceOfType FB
"Strategia sterowania Pompownia"
BEGIN
END_DATA_BLOCK

DATA_BLOCK "Write_dbHold_TCP_Sending_DB"   // DB112
VERSION : 0.1
// stored: AutoNumber true, DBAccessibleFromOPCUA true, InstanceOfName Write_dbHold_TCP_Sending, InstanceOfType FB
"Write_dbHold_TCP_Sending"
BEGIN
END_DATA_BLOCK

DATA_BLOCK "dbByte Status P1P2P3P4_DB"   // DB77
AUTHOR : rtecmer
VERSION : 0.1
// stored: AutoNumber true, DBAccessibleFromOPCUA true, InstanceOfName Byte status pomp, InstanceOfType FB
"Byte status pomp"
BEGIN
END_DATA_BLOCK

DATA_BLOCK "dbControl of   Inverters_DB"   // DB49
AUTHOR : rtecmer
VERSION : 0.1
// stored: AutoNumber true, DBAccessibleFromOPCUA true, InstanceOfName Sterowanie falownikiem, InstanceOfType FB
"Sterowanie falownikiem"
BEGIN
END_DATA_BLOCK

DATA_BLOCK "dbControl of  connection Inverters_P2"   // DB51
AUTHOR : rtecmer
VERSION : 0.1
// stored: AutoNumber true, DBAccessibleFromOPCUA true, InstanceOfName Sterowanie dołączeniem falownika, InstanceOfType FB
"Sterowanie dołączeniem falownika"
BEGIN
END_DATA_BLOCK

DATA_BLOCK "dbControl of  connection Inverters_P3"   // DB52
AUTHOR : rtecmer
VERSION : 0.1
// stored: AutoNumber true, DBAccessibleFromOPCUA true, InstanceOfName Sterowanie dołączeniem falownika, InstanceOfType FB
"Sterowanie dołączeniem falownika"
BEGIN
END_DATA_BLOCK

